LIN {X 0,Y 466.836,Z 671.645,A -85,B 0,C 180,E1 -7453.379,E2 -7453.379} C_VEL
LIN {X 0,Y 466.685,Z 675.645,A -85,B 0,C 180,E1 -7455.167,E2 -7455.167} C_VEL
LIN {X 0,Y 466.581,Z 678.329,A -85,B 0,C 180,E1 -7456.942,E2 -7456.942} C_VEL
LIN {X 0,Y 466.634,Z 679.796,A -85,B 0,C 180,E1 -7458.709,E2 -7458.709} C_VEL
LIN {X 0,Y 466.526,Z 680.097,A -85,B 0,C 180,E1 -7460.462,E2 -7460.462} C_VEL
LIN {X 0,Y 466.617,Z 679.249,A -85,B 0,C 180,E1 -7462.209,E2 -7462.209} C_VEL
LIN {X 0,Y 466.715,Z 677.258,A -85,B 0,C 180,E1 -7463.949,E2 -7463.949} C_VEL
LIN {X 0,Y 466.749,Z 674.056,A -85,B 0,C 180,E1 -7465.682,E2 -7465.682} C_VEL
LIN {X 0,Y 466.9,Z 669.606,A -85,B 0,C 180,E1 -7467.412,E2 -7467.412} C_VEL
LIN {X 0,Y 467.072,Z 663.846,A -85,B 0,C 180,E1 -7469.138,E2 -7469.138} C_VEL
LIN {X 0,Y 467.548,Z 656.595,A -85,B 0,C 180,E1 -7470.861,E2 -7470.861} C_VEL
LIN {X 0,Y 468.02,Z 648.866,A -85,B 0,C 180,E1 -7472.367,E2 -7472.367} C_VEL
LIN {X 0,Y 468.636,Z 639.619,A -85,B 0,C 180,E1 -7473.87,E2 -7473.87} C_VEL
LIN {X 0,Y 469.386,Z 628.509,A -85,B 0,C 180,E1 -7475.37,E2 -7475.37} C_VEL
LIN {X 0,Y 470.228,Z 617.061,A -85,B 0,C 180,E1 -7476.652,E2 -7476.652} C_VEL
LIN {X 0,Y 471.05,Z 604.485,A -85,B 0,C 180,E1 -7477.825,E2 -7477.825} C_VEL
LIN {X 0,Y 471.8,Z 592.099,A -85,B 0,C 180,E1 -7478.783,E2 -7478.783} C_VEL
LIN {X 0,Y 472.61,Z 578.629,A -85,B 0,C 180,E1 -7479.631,E2 -7479.631} C_VEL
LIN {X 0,Y 473.245,Z 564.922,A -85,B 0,C 180,E1 -7480.32,E2 -7480.32} C_VEL
LIN {X 0,Y 473.842,Z 550.313,A -85,B 0,C 180,E1 -7480.874,E2 -7480.874} C_VEL
LIN {X 0,Y 474.193,Z 534.838,A -85,B 0,C 180,E1 -7481.283,E2 -7481.283} C_VEL
LIN {X 0,Y 475.918,Z 391.809,A -85,B 0,C 180,E1 -7483.504,E2 -7483.504} C_VEL
LIN {X 0,Y 474.348,Z 384.081,A -85,B 0,C 180,E1 -7483.706,E2 -7483.706} C_VEL
LIN {X 0,Y 470.987,Z 371.045,A -85,B 0,C 180,E1 -7484.086,E2 -7484.086} C_VEL
LIN {X 0,Y 470.786,Z 370.175,A -85,B 0,C 180,E1 -7484.17,E2 -7484.17} C_VEL
LIN {X 0,Y 467.598,Z 355.867,A -85,B 0,C 180,E1 -7486.874,E2 -7486.874} C_VEL
LIN {X 0,Y 467.625,Z 355.863,A -85,B 0,C 180,E1 -7489.308,E2 -7489.308} C_VEL
LIN {X 0,Y 467.539,Z 355.872,A -85,B 0,C 180,E1 -7492.074,E2 -7492.074} C_VEL
LIN {X 0,Y 467.565,Z 355.866,A -85,B 0,C 180,E1 -7494.89,E2 -7494.89} C_VEL
LIN {X 0,Y 467.551,Z 355.872,A -85,B 0,C 180,E1 -7497.774,E2 -7497.774} C_VEL
LIN {X 0,Y 467.57,Z 355.865,A -85,B 0,C 180,E1 -7501.044,E2 -7501.044} C_VEL
LIN {X 0,Y 467.59,Z 355.862,A -85,B 0,C 180,E1 -7504.241,E2 -7504.241} C_VEL
LIN {X 0,Y 467.522,Z 355.869,A -85,B 0,C 180,E1 -7507.181,E2 -7507.181} C_VEL
LIN {X 0,Y 467.56,Z 355.859,A -85,B 0,C 180,E1 -7510.267,E2 -7510.267} C_VEL
LIN {X 0,Y 467.548,Z 355.87,A -85,B 0,C 180,E1 -7513.746,E2 -7513.746} C_VEL
LIN {X 0,Y 467.55,Z 355.86,A -85,B 0,C 180,E1 -7516.254,E2 -7516.254} C_VEL
LIN {X 0,Y 467.569,Z 355.864,A -85,B 0,C 180,E1 -7518.725,E2 -7518.725} C_VEL
LIN {X 0,Y 467.547,Z 355.869,A -85,B 0,C 180,E1 -7521.953,E2 -7521.953} C_VEL
LIN {X 0,Y 467.559,Z 355.868,A -85,B 0,C 180,E1 -7525.166,E2 -7525.166} C_VEL
LIN {X 0,Y 467.582,Z 355.864,A -85,B 0,C 180,E1 -7528.259,E2 -7528.259} C_VEL
LIN {X 0,Y 467.552,Z 355.866,A -85,B 0,C 180,E1 -7531.248,E2 -7531.248} C_VEL
LIN {X 0,Y 467.579,Z 355.843,A -85,B 0,C 180,E1 -7534.401,E2 -7534.401} C_VEL
LIN {X 0,Y 467.579,Z 355.857,A -85,B 0,C 180,E1 -7536.995,E2 -7536.995} C_VEL
LIN {X 0,Y 467.625,Z 355.861,A -85,B 0,C 180,E1 -7539.777,E2 -7539.777} C_VEL
LIN {X 0,Y 467.598,Z 355.852,A -85,B 0,C 180,E1 -7542.506,E2 -7542.506} C_VEL
LIN {X 0,Y 467.604,Z 355.861,A -85,B 0,C 180,E1 -7545.196,E2 -7545.196} C_VEL
LIN {X 0,Y 467.659,Z 355.848,A -85,B 0,C 180,E1 -7547.854,E2 -7547.854} C_VEL
LIN {X 0,Y 467.66,Z 355.855,A -85,B 0,C 180,E1 -7551.356,E2 -7551.356} C_VEL
LIN {X 0,Y 467.706,Z 355.842,A -85,B 0,C 180,E1 -7553.962,E2 -7553.962} C_VEL
LIN {X 0,Y 467.817,Z 355.835,A -85,B 0,C 180,E1 -7557.416,E2 -7557.416} C_VEL
LIN {X 0,Y 467.855,Z 355.826,A -85,B 0,C 180,E1 -7560,E2 -7560} C_VEL
LIN {X 0,Y 467.851,Z 355.824,A -85,B 0,C 180,E1 -7562.583,E2 -7562.583} C_VEL
LIN {X 0,Y 467.707,Z 355.847,A -85,B 0,C 180,E1 -7566.037,E2 -7566.037} C_VEL
LIN {X 0,Y 467.669,Z 355.847,A -85,B 0,C 180,E1 -7568.643,E2 -7568.643} C_VEL
LIN {X 0,Y 467.658,Z 355.849,A -85,B 0,C 180,E1 -7572.145,E2 -7572.145} C_VEL
LIN {X 0,Y 467.614,Z 355.863,A -85,B 0,C 180,E1 -7575.696,E2 -7575.696} C_VEL
LIN {X 0,Y 467.621,Z 355.857,A -85,B 0,C 180,E1 -7579.308,E2 -7579.308} C_VEL
LIN {X 0,Y 467.535,Z 355.866,A -85,B 0,C 180,E1 -7582.073,E2 -7582.073} C_VEL
LIN {X 0,Y 467.568,Z 355.863,A -85,B 0,C 180,E1 -7584.889,E2 -7584.889} C_VEL
LIN {X 0,Y 467.576,Z 355.869,A -85,B 0,C 180,E1 -7587.772,E2 -7587.772} C_VEL
LIN {X 0,Y 467.566,Z 355.865,A -85,B 0,C 180,E1 -7591.044,E2 -7591.044} C_VEL
LIN {X 0,Y 467.587,Z 355.863,A -85,B 0,C 180,E1 -7594.241,E2 -7594.241} C_VEL
LIN {X 0,Y 467.518,Z 355.872,A -85,B 0,C 180,E1 -7597.181,E2 -7597.181} C_VEL
LIN {X 0,Y 467.556,Z 355.865,A -85,B 0,C 180,E1 -7600.266,E2 -7600.266} C_VEL
LIN {X 0,Y 467.544,Z 355.873,A -85,B 0,C 180,E1 -7603.745,E2 -7603.745} C_VEL
LIN {X 0,Y 467.546,Z 355.869,A -85,B 0,C 180,E1 -7606.254,E2 -7606.254} C_VEL
LIN {X 0,Y 467.565,Z 355.866,A -85,B 0,C 180,E1 -7608.725,E2 -7608.725} C_VEL
LIN {X 0,Y 467.546,Z 355.871,A -85,B 0,C 180,E1 -7611.953,E2 -7611.953} C_VEL
LIN {X 0,Y 467.555,Z 355.87,A -85,B 0,C 180,E1 -7615.166,E2 -7615.166} C_VEL
LIN {X 0,Y 467.582,Z 355.866,A -85,B 0,C 180,E1 -7618.26,E2 -7618.26} C_VEL
LIN {X 0,Y 467.625,Z 356.033,A -85,B 0,C 180,E1 -7619.676,E2 -7619.676} C_VEL
LIN {X 0,Y 471.614,Z 372.945,A -85,B 0,C 180,E1 -7622.486,E2 -7622.486} C_VEL
LIN {X 0,Y 472.119,Z 377.049,A -85,B 0,C 180,E1 -7623.129,E2 -7623.129} C_VEL
LIN {X 0,Y 471.109,Z 396.315,A -85,B 0,C 180,E1 -7625.931,E2 -7625.931} C_VEL
LIN {X 0,Y 475.766,Z 421.055,A -85,B 0,C 180,E1 -7626.562,E2 -7626.562} C_VEL
LIN {X 0,Y 474.108,Z 562.68,A -85,B 0,C 180,E1 -7628.761,E2 -7628.761} C_VEL
LIN {X 0,Y 473.524,Z 578.617,A -85,B 0,C 180,E1 -7629.18,E2 -7629.18} C_VEL
LIN {X 0,Y 472.879,Z 594.115,A -85,B 0,C 180,E1 -7629.783,E2 -7629.783} C_VEL
LIN {X 0,Y 472.107,Z 608.851,A -85,B 0,C 180,E1 -7630.544,E2 -7630.544} C_VEL
LIN {X 0,Y 471.355,Z 622.223,A -85,B 0,C 180,E1 -7631.415,E2 -7631.415} C_VEL
LIN {X 0,Y 470.411,Z 635.801,A -85,B 0,C 180,E1 -7632.502,E2 -7632.502} C_VEL
LIN {X 0,Y 469.599,Z 648.146,A -85,B 0,C 180,E1 -7633.703,E2 -7633.703} C_VEL
LIN {X 0,Y 468.814,Z 659.403,A -85,B 0,C 180,E1 -7635.013,E2 -7635.013} C_VEL
LIN {X 0,Y 468.143,Z 670.327,A -85,B 0,C 180,E1 -7636.544,E2 -7636.544} C_VEL
LIN {X 0,Y 467.603,Z 679.411,A -85,B 0,C 180,E1 -7638.073,E2 -7638.073} C_VEL
LIN {X 0,Y 467.234,Z 686.944,A -85,B 0,C 180,E1 -7639.601,E2 -7639.601} C_VEL
LIN {X 0,Y 466.935,Z 693.971,A -85,B 0,C 180,E1 -7641.343,E2 -7641.343} C_VEL
LIN {X 0,Y 466.818,Z 699.495,A -85,B 0,C 180,E1 -7643.082,E2 -7643.082} C_VEL
LIN {X 0,Y 466.686,Z 703.668,A -85,B 0,C 180,E1 -7644.816,E2 -7644.816} C_VEL
LIN {X 0,Y 466.671,Z 706.594,A -85,B 0,C 180,E1 -7646.546,E2 -7646.546} C_VEL
LIN {X 0,Y 466.628,Z 708.336,A -85,B 0,C 180,E1 -7648.274,E2 -7648.274} C_VEL
LIN {X 0,Y 466.595,Z 708.93,A -85,B 0,C 180,E1 -7650,E2 -7650} C_VEL
LIN {X 0,Y 466.628,Z 708.325,A -85,B 0,C 180,E1 -7651.726,E2 -7651.726} C_VEL
LIN {X 0,Y 466.671,Z 706.573,A -85,B 0,C 180,E1 -7653.454,E2 -7653.454} C_VEL
LIN {X 0,Y 466.684,Z 703.644,A -85,B 0,C 180,E1 -7655.184,E2 -7655.184} C_VEL
LIN {X 0,Y 466.74,Z 699.47,A -85,B 0,C 180,E1 -7656.919,E2 -7656.919} C_VEL
LIN {X 0,Y 466.934,Z 693.945,A -85,B 0,C 180,E1 -7658.657,E2 -7658.657} C_VEL
LIN {X 0,Y 467.234,Z 686.922,A -85,B 0,C 180,E1 -7660.399,E2 -7660.399} C_VEL
LIN {X 0,Y 467.633,Z 679.411,A -85,B 0,C 180,E1 -7661.926,E2 -7661.926} C_VEL
LIN {X 0,Y 468.135,Z 670.368,A -85,B 0,C 180,E1 -7663.456,E2 -7663.456} C_VEL
LIN {X 0,Y 468.843,Z 659.518,A -85,B 0,C 180,E1 -7664.986,E2 -7664.986} C_VEL
LIN {X 0,Y 469.735,Z 647.346,A -85,B 0,C 180,E1 -7666.404,E2 -7666.404} C_VEL
LIN {X 0,Y 470.532,Z 634.953,A -85,B 0,C 180,E1 -7667.605,E2 -7667.605} C_VEL
LIN {X 0,Y 471.468,Z 621.272,A -85,B 0,C 180,E1 -7668.693,E2 -7668.693} C_VEL
LIN {X 0,Y 472.291,Z 607.87,A -85,B 0,C 180,E1 -7669.561,E2 -7669.561} C_VEL
LIN {X 0,Y 473.095,Z 593.523,A -85,B 0,C 180,E1 -7670.298,E2 -7670.298} C_VEL
LIN {X 0,Y 473.713,Z 578.414,A -85,B 0,C 180,E1 -7670.887,E2 -7670.887} C_VEL
LIN {X 0,Y 474.286,Z 562.15,A -85,B 0,C 180,E1 -7671.316,E2 -7671.316} C_VEL
LIN {X 0,Y 476.029,Z 420.259,A -85,B 0,C 180,E1 -7673.546,E2 -7673.546} C_VEL
LIN {X 0,Y 471.305,Z 396.045,A -85,B 0,C 180,E1 -7674.228,E2 -7674.228} C_VEL
LIN {X 0,Y 472.463,Z 377.157,A -85,B 0,C 180,E1 -7677.034,E2 -7677.034} C_VEL
LIN {X 0,Y 471.018,Z 369.489,A -85,B 0,C 180,E1 -7678.318,E2 -7678.318} C_VEL
LIN {X 0,Y 467.576,Z 355.874,A -85,B 0,C 180,E1 -7680.733,E2 -7680.733} C_VEL
LIN {X 0,Y 467.568,Z 355.869,A -85,B 0,C 180,E1 -7683.79,E2 -7683.79} C_VEL
LIN {X 0,Y 467.517,Z 355.874,A -85,B 0,C 180,E1 -7686.963,E2 -7686.963} C_VEL
LIN {X 0,Y 467.557,Z 355.87,A -85,B 0,C 180,E1 -7690.267,E2 -7690.267} C_VEL
LIN {X 0,Y 467.542,Z 355.869,A -85,B 0,C 180,E1 -7692.566,E2 -7692.566} C_VEL
LIN {X 0,Y 467.564,Z 355.867,A -85,B 0,C 180,E1 -7695.053,E2 -7695.053} C_VEL
LIN {X 0,Y 467.56,Z 355.87,A -85,B 0,C 180,E1 -7698.726,E2 -7698.726} C_VEL
LIN {X 0,Y 467.543,Z 355.87,A -85,B 0,C 180,E1 -7701.954,E2 -7701.954} C_VEL
LIN {X 0,Y 467.561,Z 355.863,A -85,B 0,C 180,E1 -7705.167,E2 -7705.167} C_VEL
LIN {X 0,Y 467.582,Z 355.857,A -85,B 0,C 180,E1 -7708.26,E2 -7708.26} C_VEL
LIN {X 0,Y 467.555,Z 355.864,A -85,B 0,C 180,E1 -7711.249,E2 -7711.249} C_VEL
LIN {X 0,Y 467.582,Z 355.863,A -85,B 0,C 180,E1 -7714.159,E2 -7714.159} C_VEL
LIN {X 0,Y 467.576,Z 355.862,A -85,B 0,C 180,E1 -7716.996,E2 -7716.996} C_VEL
LIN {X 0,Y 467.621,Z 355.858,A -85,B 0,C 180,E1 -7719.777,E2 -7719.777} C_VEL
LIN {X 0,Y 467.589,Z 355.867,A -85,B 0,C 180,E1 -7722.506,E2 -7722.506} C_VEL
LIN {X 0,Y 467.6,Z 355.86,A -85,B 0,C 180,E1 -7725.197,E2 -7725.197} C_VEL
LIN {X 0,Y 467.658,Z 355.851,A -85,B 0,C 180,E1 -7727.855,E2 -7727.855} C_VEL
LIN {X 0,Y 467.668,Z 355.848,A -85,B 0,C 180,E1 -7731.357,E2 -7731.357} C_VEL
LIN {X 0,Y 467.714,Z 355.848,A -85,B 0,C 180,E1 -7733.963,E2 -7733.963} C_VEL
LIN {X 0,Y 467.852,Z 355.829,A -85,B 0,C 180,E1 -7737.417,E2 -7737.417} C_VEL
LIN {X 0,Y 467.854,Z 355.826,A -85,B 0,C 180,E1 -7740,E2 -7740} C_VEL
LIN {X 0,Y 467.848,Z 355.831,A -85,B 0,C 180,E1 -7742.583,E2 -7742.583} C_VEL
LIN {X 0,Y 467.714,Z 355.849,A -85,B 0,C 180,E1 -7746.038,E2 -7746.038} C_VEL
LIN {X 0,Y 467.666,Z 355.858,A -85,B 0,C 180,E1 -7748.643,E2 -7748.643} C_VEL
LIN {X 0,Y 467.659,Z 355.854,A -85,B 0,C 180,E1 -7752.146,E2 -7752.146} C_VEL
LIN {X 0,Y 467.642,Z 355.854,A -85,B 0,C 180,E1 -7755.695,E2 -7755.695} C_VEL
LIN {X 0,Y 467.624,Z 355.843,A -85,B 0,C 180,E1 -7759.308,E2 -7759.308} C_VEL
LIN {X 0,Y 467.538,Z 355.868,A -85,B 0,C 180,E1 -7762.074,E2 -7762.074} C_VEL
LIN {X 0,Y 467.563,Z 355.856,A -85,B 0,C 180,E1 -7764.89,E2 -7764.89} C_VEL
LIN {X 0,Y 467.582,Z 355.862,A -85,B 0,C 180,E1 -7767.772,E2 -7767.772} C_VEL
LIN {X 0,Y 467.571,Z 355.857,A -85,B 0,C 180,E1 -7771.045,E2 -7771.045} C_VEL
LIN {X 0,Y 467.58,Z 355.868,A -85,B 0,C 180,E1 -7774.24,E2 -7774.24} C_VEL
LIN {X 0,Y 467.526,Z 355.872,A -85,B 0,C 180,E1 -7777.182,E2 -7777.182} C_VEL
LIN {X 0,Y 467.561,Z 355.865,A -85,B 0,C 180,E1 -7780.267,E2 -7780.267} C_VEL
LIN {X 0,Y 467.55,Z 355.869,A -85,B 0,C 180,E1 -7783.746,E2 -7783.746} C_VEL
LIN {X 0,Y 467.552,Z 355.869,A -85,B 0,C 180,E1 -7786.255,E2 -7786.255} C_VEL
LIN {X 0,Y 467.574,Z 355.867,A -85,B 0,C 180,E1 -7789.735,E2 -7789.735} C_VEL
LIN {X 0,Y 467.565,Z 355.969,A -85,B 0,C 180,E1 -7792.929,E2 -7792.929} C_VEL
LIN {X 0,Y 470.544,Z 368.645,A -85,B 0,C 180,E1 -7795.419,E2 -7795.419} C_VEL
LIN {X 0,Y 470.999,Z 370.7,A -85,B 0,C 180,E1 -7795.813,E2 -7795.813} C_VEL
LIN {X 0,Y 473.185,Z 377.561,A -85,B 0,C 180,E1 -7796.064,E2 -7796.064} C_VEL
LIN {X 0,Y 476.317,Z 391.74,A -85,B 0,C 180,E1 -7796.479,E2 -7796.479} C_VEL
LIN {X 0,Y 474.65,Z 517.95,A -85,B 0,C 180,E1 -7798.444,E2 -7798.444} C_VEL
LIN {X 0,Y 473.931,Z 523.804,A -85,B 0,C 180,E1 -7798.5,E2 -7798.5} C_VEL
LIN {X 0,Y 468.73,Z 540.884,A -85,B 0,C 180,E1 -7798.579,E2 -7798.579} C_VEL
LIN {X 0,Y 467.607,Z 546.618,A -85,B 0,C 180,E1 -7798.686,E2 -7798.686} C_VEL
LIN {X 0,Y 467.497,Z 548.534,A -85,B 0,C 180,E1 -7798.742,E2 -7798.742} C_VEL
LIN {X 0,Y 466.936,Z 563.073,A -85,B 0,C 180,E1 -7799.283,E2 -7799.283} C_VEL
LIN {X 0,Y 466.171,Z 577.184,A -85,B 0,C 180,E1 -7799.978,E2 -7799.978} C_VEL
LIN {X 0,Y 465.384,Z 591.094,A -85,B 0,C 180,E1 -7800.855,E2 -7800.855} C_VEL
LIN {X 0,Y 464.463,Z 604.731,A -85,B 0,C 180,E1 -7801.919,E2 -7801.919} C_VEL
LIN {X 0,Y 463.464,Z 617.402,A -85,B 0,C 180,E1 -7803.124,E2 -7803.124} C_VEL
LIN {X 0,Y 462.676,Z 628.129,A -85,B 0,C 180,E1 -7804.347,E2 -7804.347} C_VEL
LIN {X 0,Y 461.84,Z 638.445,A -85,B 0,C 180,E1 -7805.741,E2 -7805.741} C_VEL
LIN {X 0,Y 461.203,Z 647.16,A -85,B 0,C 180,E1 -7807.134,E2 -7807.134} C_VEL
LIN {X 0,Y 460.644,Z 655.619,A -85,B 0,C 180,E1 -7808.755,E2 -7808.755} C_VEL
LIN {X 0,Y 460.167,Z 662.538,A -85,B 0,C 180,E1 -7810.367,E2 -7810.367} C_VEL
LIN {X 0,Y 459.897,Z 668.876,A -85,B 0,C 180,E1 -7812.204,E2 -7812.204} C_VEL
LIN {X 0,Y 459.73,Z 673.684,A -85,B 0,C 180,E1 -7814.028,E2 -7814.028} C_VEL
LIN {X 0,Y 459.526,Z 677.12,A -85,B 0,C 180,E1 -7815.836,E2 -7815.836} C_VEL
LIN {X 0,Y 459.522,Z 679.296,A -85,B 0,C 180,E1 -7817.636,E2 -7817.636} C_VEL
LIN {X 0,Y 459.492,Z 680.282,A -85,B 0,C 180,E1 -7819.424,E2 -7819.424} C_VEL
LIN {X 0,Y 459.457,Z 680.115,A -85,B 0,C 180,E1 -7821.201,E2 -7821.201} C_VEL
LIN {X 0,Y 459.573,Z 678.794,A -85,B 0,C 180,E1 -7822.973,E2 -7822.973} C_VEL
LIN {X 0,Y 459.642,Z 676.271,A -85,B 0,C 180,E1 -7824.736,E2 -7824.736} C_VEL
LIN {X 0,Y 459.799,Z 672.548,A -85,B 0,C 180,E1 -7826.495,E2 -7826.495} C_VEL
LIN {X 0,Y 459.844,Z 667.581,A -85,B 0,C 180,E1 -7828.248,E2 -7828.248} C_VEL
LIN {X 0,Y 460.263,Z 661.209,A -85,B 0,C 180,E1 -7830,E2 -7830} C_VEL
LIN {X 0,Y 460.738,Z 653.281,A -85,B 0,C 180,E1 -7831.748,E2 -7831.748} C_VEL
LIN {X 0,Y 461.37,Z 644.846,A -85,B 0,C 180,E1 -7833.275,E2 -7833.275} C_VEL
LIN {X 0,Y 462.046,Z 634.757,A -85,B 0,C 180,E1 -7834.799,E2 -7834.799} C_VEL
LIN {X 0,Y 462.806,Z 624.46,A -85,B 0,C 180,E1 -7836.102,E2 -7836.102} C_VEL
LIN {X 0,Y 463.689,Z 613.277,A -85,B 0,C 180,E1 -7837.293,E2 -7837.293} C_VEL
LIN {X 0,Y 464.494,Z 601.199,A -85,B 0,C 180,E1 -7838.374,E2 -7838.374} C_VEL
LIN {X 0,Y 465.4,Z 588.004,A -85,B 0,C 180,E1 -7839.343,E2 -7839.343} C_VEL
LIN {X 0,Y 466.146,Z 573.447,A -85,B 0,C 180,E1 -7840.204,E2 -7840.204} C_VEL
LIN {X 0,Y 466.792,Z 559.337,A -85,B 0,C 180,E1 -7840.848,E2 -7840.848} C_VEL
LIN {X 0,Y 467.353,Z 544.154,A -85,B 0,C 180,E1 -7841.356,E2 -7841.356} C_VEL
LIN {X 0,Y 467.695,Z 529.518,A -85,B 0,C 180,E1 -7841.677,E2 -7841.677} C_VEL
LIN {X 0,Y 469.285,Z 391.719,A -85,B 0,C 180,E1 -7843.836,E2 -7843.836} C_VEL
LIN {X 0,Y 464.953,Z 374.167,A -85,B 0,C 180,E1 -7844.345,E2 -7844.345} C_VEL
LIN {X 0,Y 463.682,Z 370.698,A -85,B 0,C 180,E1 -7844.481,E2 -7844.481} C_VEL
LIN {X 0,Y 460.55,Z 356.745,A -85,B 0,C 180,E1 -7847.14,E2 -7847.14} C_VEL
LIN {X 0,Y 460.572,Z 356.742,A -85,B 0,C 180,E1 -7849.615,E2 -7849.615} C_VEL
LIN {X 0,Y 460.515,Z 356.745,A -85,B 0,C 180,E1 -7852.429,E2 -7852.429} C_VEL
LIN {X 0,Y 460.539,Z 356.745,A -85,B 0,C 180,E1 -7855.793,E2 -7855.793} C_VEL
LIN {X 0,Y 460.525,Z 356.745,A -85,B 0,C 180,E1 -7859.232,E2 -7859.232} C_VEL
LIN {X 0,Y 460.535,Z 356.736,A -85,B 0,C 180,E1 -7862.284,E2 -7862.284} C_VEL
LIN {X 0,Y 460.508,Z 356.747,A -85,B 0,C 180,E1 -7865.446,E2 -7865.446} C_VEL
LIN {X 0,Y 460.497,Z 356.746,A -85,B 0,C 180,E1 -7868.889,E2 -7868.889} C_VEL
LIN {X 0,Y 460.506,Z 356.745,A -85,B 0,C 180,E1 -7871.598,E2 -7871.598} C_VEL
LIN {X 0,Y 460.515,Z 356.74,A -85,B 0,C 180,E1 -7874.589,E2 -7874.589} C_VEL
LIN {X 0,Y 460.495,Z 356.75,A -85,B 0,C 180,E1 -7877.815,E2 -7877.815} C_VEL
LIN {X 0,Y 460.514,Z 356.742,A -85,B 0,C 180,E1 -7880.135,E2 -7880.135} C_VEL
LIN {X 0,Y 460.469,Z 356.755,A -85,B 0,C 180,E1 -7883.469,E2 -7883.469} C_VEL
LIN {X 0,Y 460.52,Z 356.74,A -85,B 0,C 180,E1 -7886.674,E2 -7886.674} C_VEL
LIN {X 0,Y 460.51,Z 356.745,A -85,B 0,C 180,E1 -7889.759,E2 -7889.759} C_VEL
LIN {X 0,Y 460.494,Z 356.729,A -85,B 0,C 180,E1 -7892.751,E2 -7892.751} C_VEL
LIN {X 0,Y 460.52,Z 356.732,A -85,B 0,C 180,E1 -7895.666,E2 -7895.666} C_VEL
LIN {X 0,Y 460.525,Z 356.741,A -85,B 0,C 180,E1 -7898.578,E2 -7898.578} C_VEL
LIN {X 0,Y 460.588,Z 356.737,A -85,B 0,C 180,E1 -7901.31,E2 -7901.31} C_VEL
LIN {X 0,Y 460.608,Z 356.732,A -85,B 0,C 180,E1 -7904.059,E2 -7904.059} C_VEL
LIN {X 0,Y 460.613,Z 356.728,A -85,B 0,C 180,E1 -7907.665,E2 -7907.665} C_VEL
LIN {X 0,Y 460.612,Z 356.731,A -85,B 0,C 180,E1 -7911.223,E2 -7911.223} C_VEL
LIN {X 0,Y 460.672,Z 356.719,A -85,B 0,C 180,E1 -7913.869,E2 -7913.869} C_VEL
LIN {X 0,Y 460.761,Z 356.714,A -85,B 0,C 180,E1 -7917.377,E2 -7917.377} C_VEL
LIN {X 0,Y 460.824,Z 356.702,A -85,B 0,C 180,E1 -7920,E2 -7920} C_VEL
LIN {X 0,Y 460.791,Z 356.703,A -85,B 0,C 180,E1 -7922.622,E2 -7922.622} C_VEL
LIN {X 0,Y 460.673,Z 356.722,A -85,B 0,C 180,E1 -7926.13,E2 -7926.13} C_VEL
LIN {X 0,Y 460.619,Z 356.726,A -85,B 0,C 180,E1 -7928.776,E2 -7928.776} C_VEL
LIN {X 0,Y 460.599,Z 356.727,A -85,B 0,C 180,E1 -7932.435,E2 -7932.435} C_VEL
LIN {X 0,Y 460.558,Z 356.738,A -85,B 0,C 180,E1 -7935.978,E2 -7935.978} C_VEL
LIN {X 0,Y 460.568,Z 356.74,A -85,B 0,C 180,E1 -7939.615,E2 -7939.615} C_VEL
LIN {X 0,Y 460.511,Z 356.738,A -85,B 0,C 180,E1 -7942.428,E2 -7942.428} C_VEL
LIN {X 0,Y 460.536,Z 356.742,A -85,B 0,C 180,E1 -7945.793,E2 -7945.793} C_VEL
LIN {X 0,Y 460.521,Z 356.743,A -85,B 0,C 180,E1 -7948.235,E2 -7948.235} C_VEL
LIN {X 0,Y 460.52,Z 356.745,A -85,B 0,C 180,E1 -7951.282,E2 -7951.282} C_VEL
LIN {X 0,Y 460.529,Z 356.741,A -85,B 0,C 180,E1 -7954.504,E2 -7954.504} C_VEL
LIN {X 0,Y 460.483,Z 356.752,A -85,B 0,C 180,E1 -7957.625,E2 -7957.625} C_VEL
LIN {X 0,Y 460.515,Z 356.742,A -85,B 0,C 180,E1 -7961.013,E2 -7961.013} C_VEL
LIN {X 0,Y 460.51,Z 356.743,A -85,B 0,C 180,E1 -7964.589,E2 -7964.589} C_VEL
LIN {X 0,Y 460.49,Z 356.753,A -85,B 0,C 180,E1 -7967.815,E2 -7967.815} C_VEL
LIN {X 0,Y 460.51,Z 356.749,A -85,B 0,C 180,E1 -7970.135,E2 -7970.135} C_VEL
LIN {X 0,Y 460.465,Z 356.757,A -85,B 0,C 180,E1 -7973.469,E2 -7973.469} C_VEL
LIN {X 0,Y 460.519,Z 356.745,A -85,B 0,C 180,E1 -7976.674,E2 -7976.674} C_VEL
LIN {X 0,Y 460.556,Z 356.767,A -85,B 0,C 180,E1 -7979.351,E2 -7979.351} C_VEL
LIN {X 0,Y 464.667,Z 374.114,A -85,B 0,C 180,E1 -7982.284,E2 -7982.284} C_VEL
LIN {X 0,Y 465.272,Z 377.365,A -85,B 0,C 180,E1 -7982.811,E2 -7982.811} C_VEL
LIN {X 0,Y 464.289,Z 396.076,A -85,B 0,C 180,E1 -7985.579,E2 -7985.579} C_VEL
LIN {X 0,Y 469.164,Z 422.584,A -85,B 0,C 180,E1 -7986.263,E2 -7986.263} C_VEL
LIN {X 0,Y 467.421,Z 562.843,A -85,B 0,C 180,E1 -7988.471,E2 -7988.471} C_VEL
LIN {X 0,Y 466.819,Z 578.838,A -85,B 0,C 180,E1 -7988.904,E2 -7988.904} C_VEL
LIN {X 0,Y 466.169,Z 593.903,A -85,B 0,C 180,E1 -7989.498,E2 -7989.498} C_VEL
LIN {X 0,Y 465.368,Z 608.345,A -85,B 0,C 180,E1 -7990.25,E2 -7990.25} C_VEL
LIN {X 0,Y 464.533,Z 621.77,A -85,B 0,C 180,E1 -7991.132,E2 -7991.132} C_VEL
LIN {X 0,Y 463.564,Z 635.41,A -85,B 0,C 180,E1 -7992.235,E2 -7992.235} C_VEL
LIN {X 0,Y 462.727,Z 647.794,A -85,B 0,C 180,E1 -7993.454,E2 -7993.454} C_VEL
LIN {X 0,Y 461.881,Z 659.078,A -85,B 0,C 180,E1 -7994.783,E2 -7994.783} C_VEL
LIN {X 0,Y 461.167,Z 670.036,A -85,B 0,C 180,E1 -7996.337,E2 -7996.337} C_VEL
LIN {X 0,Y 460.58,Z 679.136,A -85,B 0,C 180,E1 -7997.889,E2 -7997.889} C_VEL
LIN {X 0,Y 460.213,Z 686.683,A -85,B 0,C 180,E1 -7999.441,E2 -7999.441} C_VEL
LIN {X 0,Y 459.873,Z 693.725,A -85,B 0,C 180,E1 -8001.209,E2 -8001.209} C_VEL
LIN {X 0,Y 459.727,Z 699.259,A -85,B 0,C 180,E1 -8002.975,E2 -8002.975} C_VEL
LIN {X 0,Y 459.597,Z 703.44,A -85,B 0,C 180,E1 -8004.736,E2 -8004.736} C_VEL
LIN {X 0,Y 459.565,Z 706.37,A -85,B 0,C 180,E1 -8006.493,E2 -8006.493} C_VEL
LIN {X 0,Y 459.539,Z 708.116,A -85,B 0,C 180,E1 -8008.247,E2 -8008.247} C_VEL
LIN {X 0,Y 459.527,Z 708.712,A -85,B 0,C 180,E1 -8010,E2 -8010} C_VEL
LIN {X 0,Y 459.539,Z 708.108,A -85,B 0,C 180,E1 -8011.753,E2 -8011.753} C_VEL
LIN {X 0,Y 459.565,Z 706.358,A -85,B 0,C 180,E1 -8013.507,E2 -8013.507} C_VEL
LIN {X 0,Y 459.594,Z 703.433,A -85,B 0,C 180,E1 -8015.264,E2 -8015.264} C_VEL
LIN {X 0,Y 459.662,Z 699.265,A -85,B 0,C 180,E1 -8017.026,E2 -8017.026} C_VEL
LIN {X 0,Y 459.872,Z 693.751,A -85,B 0,C 180,E1 -8018.791,E2 -8018.791} C_VEL
LIN {X 0,Y 460.212,Z 686.741,A -85,B 0,C 180,E1 -8020.559,E2 -8020.559} C_VEL
LIN {X 0,Y 460.604,Z 679.242,A -85,B 0,C 180,E1 -8022.111,E2 -8022.111} C_VEL
LIN {X 0,Y 461.155,Z 670.22,A -85,B 0,C 180,E1 -8023.664,E2 -8023.664} C_VEL
LIN {X 0,Y 461.903,Z 659.397,A -85,B 0,C 180,E1 -8025.216,E2 -8025.216} C_VEL
LIN {X 0,Y 462.873,Z 647.272,A -85,B 0,C 180,E1 -8026.654,E2 -8026.654} C_VEL
LIN {X 0,Y 463.721,Z 634.921,A -85,B 0,C 180,E1 -8027.873,E2 -8027.873} C_VEL
LIN {X 0,Y 464.729,Z 621.305,A -85,B 0,C 180,E1 -8028.974,E2 -8028.974} C_VEL
LIN {X 0,Y 465.602,Z 607.964,A -85,B 0,C 180,E1 -8029.854,E2 -8029.854} C_VEL
LIN {X 0,Y 466.498,Z 592.589,A -85,B 0,C 180,E1 -8030.653,E2 -8030.653} C_VEL
LIN {X 0,Y 467.18,Z 577.109,A -85,B 0,C 180,E1 -8031.251,E2 -8031.251} C_VEL
LIN {X 0,Y 467.756,Z 561.566,A -85,B 0,C 180,E1 -8031.657,E2 -8031.657} C_VEL
LIN {X 0,Y 469.597,Z 421.323,A -85,B 0,C 180,E1 -8033.892,E2 -8033.892} C_VEL
LIN {X 0,Y 464.555,Z 395.836,A -85,B 0,C 180,E1 -8034.63,E2 -8034.63} C_VEL
LIN {X 0,Y 465.693,Z 379.057,A -85,B 0,C 180,E1 -8037.162,E2 -8037.162} C_VEL
LIN {X 0,Y 463.951,Z 370.166,A -85,B 0,C 180,E1 -8038.686,E2 -8038.686} C_VEL
LIN {X 0,Y 461.136,Z 359.008,A -85,B 0,C 180,E1 -8040.701,E2 -8040.701} C_VEL
LIN {X 0,Y 460.535,Z 356.745,A -85,B 0,C 180,E1 -8041.128,E2 -8041.128} C_VEL
LIN {X 0,Y 460.521,Z 356.748,A -85,B 0,C 180,E1 -8044.504,E2 -8044.504} C_VEL
LIN {X 0,Y 460.491,Z 356.748,A -85,B 0,C 180,E1 -8047.624,E2 -8047.624} C_VEL
LIN {X 0,Y 460.517,Z 356.742,A -85,B 0,C 180,E1 -8051.013,E2 -8051.013} C_VEL
LIN {X 0,Y 460.51,Z 356.749,A -85,B 0,C 180,E1 -8054.589,E2 -8054.589} C_VEL
LIN {X 0,Y 460.478,Z 356.75,A -85,B 0,C 180,E1 -8057.814,E2 -8057.814} C_VEL
LIN {X 0,Y 460.509,Z 356.748,A -85,B 0,C 180,E1 -8060.136,E2 -8060.136} C_VEL
LIN {X 0,Y 460.465,Z 356.74,A -85,B 0,C 180,E1 -8063.47,E2 -8063.47} C_VEL
LIN {X 0,Y 460.529,Z 356.743,A -85,B 0,C 180,E1 -8066.675,E2 -8066.675} C_VEL
LIN {X 0,Y 460.506,Z 356.731,A -85,B 0,C 180,E1 -8069.76,E2 -8069.76} C_VEL
LIN {X 0,Y 460.533,Z 356.741,A -85,B 0,C 180,E1 -8072.754,E2 -8072.754} C_VEL
LIN {X 0,Y 460.521,Z 356.743,A -85,B 0,C 180,E1 -8075.667,E2 -8075.667} C_VEL
LIN {X 0,Y 460.522,Z 356.748,A -85,B 0,C 180,E1 -8078.579,E2 -8078.579} C_VEL
LIN {X 0,Y 460.584,Z 356.733,A -85,B 0,C 180,E1 -8081.311,E2 -8081.311} C_VEL
LIN {X 0,Y 460.586,Z 356.735,A -85,B 0,C 180,E1 -8084.059,E2 -8084.059} C_VEL
LIN {X 0,Y 460.611,Z 356.728,A -85,B 0,C 180,E1 -8087.666,E2 -8087.666} C_VEL
LIN {X 0,Y 460.619,Z 356.726,A -85,B 0,C 180,E1 -8091.224,E2 -8091.224} C_VEL
LIN {X 0,Y 460.679,Z 356.724,A -85,B 0,C 180,E1 -8093.87,E2 -8093.87} C_VEL
LIN {X 0,Y 460.792,Z 356.708,A -85,B 0,C 180,E1 -8097.378,E2 -8097.378} C_VEL
LIN {X 0,Y 460.824,Z 356.702,A -85,B 0,C 180,E1 -8100,E2 -8100} C_VEL
LIN {X 0,Y 460.788,Z 356.71,A -85,B 0,C 180,E1 -8102.623,E2 -8102.623} C_VEL
LIN {X 0,Y 460.678,Z 356.726,A -85,B 0,C 180,E1 -8106.131,E2 -8106.131} C_VEL
LIN {X 0,Y 460.617,Z 356.734,A -85,B 0,C 180,E1 -8108.777,E2 -8108.777} C_VEL
LIN {X 0,Y 460.616,Z 356.735,A -85,B 0,C 180,E1 -8112.445,E2 -8112.445} C_VEL
LIN {X 0,Y 460.603,Z 356.733,A -85,B 0,C 180,E1 -8115.998,E2 -8115.998} C_VEL
LIN {X 0,Y 460.57,Z 356.721,A -85,B 0,C 180,E1 -8119.616,E2 -8119.616} C_VEL
LIN {X 0,Y 460.514,Z 356.748,A -85,B 0,C 180,E1 -8122.429,E2 -8122.429} C_VEL
LIN {X 0,Y 460.537,Z 356.728,A -85,B 0,C 180,E1 -8125.794,E2 -8125.794} C_VEL
LIN {X 0,Y 460.528,Z 356.744,A -85,B 0,C 180,E1 -8128.235,E2 -8128.235} C_VEL
LIN {X 0,Y 460.524,Z 356.735,A -85,B 0,C 180,E1 -8131.283,E2 -8131.283} C_VEL
LIN {X 0,Y 460.525,Z 356.741,A -85,B 0,C 180,E1 -8134.504,E2 -8134.504} C_VEL
LIN {X 0,Y 460.489,Z 356.747,A -85,B 0,C 180,E1 -8137.625,E2 -8137.625} C_VEL
LIN {X 0,Y 460.521,Z 356.745,A -85,B 0,C 180,E1 -8141.013,E2 -8141.013} C_VEL
LIN {X 0,Y 460.515,Z 356.746,A -85,B 0,C 180,E1 -8144.59,E2 -8144.59} C_VEL
LIN {X 0,Y 460.508,Z 356.743,A -85,B 0,C 180,E1 -8147.817,E2 -8147.817} C_VEL
LIN {X 0,Y 460.523,Z 356.748,A -85,B 0,C 180,E1 -8150.137,E2 -8150.137} C_VEL
LIN {X 0,Y 460.508,Z 356.834,A -85,B 0,C 180,E1 -8152.557,E2 -8152.557} C_VEL
LIN {X 0,Y 463.625,Z 369.899,A -85,B 0,C 180,E1 -8155.177,E2 -8155.177} C_VEL
LIN {X 0,Y 463.923,Z 371.197,A -85,B 0,C 180,E1 -8155.397,E2 -8155.397} C_VEL
LIN {X 0,Y 466.741,Z 378.624,A -85,B 0,C 180,E1 -8155.697,E2 -8155.697} C_VEL
LIN {X 0,Y 469.834,Z 392.084,A -85,B 0,C 180,E1 -8156.108,E2 -8156.108} C_VEL
LIN {X 0,Y 468.092,Z 520.515,A -85,B 0,C 180,E1 -8158.14,E2 -8158.14} C_VEL
LIN {X 0,Y 467.825,Z 539.358,A -85,B 0,C 180,E1 -8158.492,E2 -8158.492} C_VEL
LIN {X 0,Y 467.497,Z 548.534,A -85,B 0,C 180,E1 -8158.742,E2 -8158.742} C_VEL
LIN {X 0,Y 466.667,Z 554.254,A -85,B 0,C 180,E1 -8158.898,E2 -8158.898} C_VEL
LIN {X 0,Y 463.605,Z 563.513,A -85,B 0,C 180,E1 -8159.126,E2 -8159.126} C_VEL
LIN {X 0,Y 460.477,Z 572.639,A -85,B 0,C 180,E1 -8159.422,E2 -8159.422} C_VEL
LIN {X 0,Y 459.538,Z 578.009,A -85,B 0,C 180,E1 -8159.686,E2 -8159.686} C_VEL
LIN {X 0,Y 458.76,Z 591.001,A -85,B 0,C 180,E1 -8160.519,E2 -8160.519} C_VEL
LIN {X 0,Y 457.777,Z 604.5,A -85,B 0,C 180,E1 -8161.58,E2 -8161.58} C_VEL
LIN {X 0,Y 456.781,Z 616.656,A -85,B 0,C 180,E1 -8162.74,E2 -8162.74} C_VEL
LIN {X 0,Y 455.936,Z 627.219,A -85,B 0,C 180,E1 -8163.94,E2 -8163.94} C_VEL
LIN {X 0,Y 455.051,Z 637.721,A -85,B 0,C 180,E1 -8165.355,E2 -8165.355} C_VEL
LIN {X 0,Y 454.35,Z 646.543,A -85,B 0,C 180,E1 -8166.769,E2 -8166.769} C_VEL
LIN {X 0,Y 453.764,Z 654.697,A -85,B 0,C 180,E1 -8168.327,E2 -8168.327} C_VEL
LIN {X 0,Y 453.192,Z 662.174,A -85,B 0,C 180,E1 -8170.052,E2 -8170.052} C_VEL
LIN {X 0,Y 452.869,Z 668.633,A -85,B 0,C 180,E1 -8171.918,E2 -8171.918} C_VEL
LIN {X 0,Y 452.649,Z 673.558,A -85,B 0,C 180,E1 -8173.771,E2 -8173.771} C_VEL
LIN {X 0,Y 452.474,Z 677.104,A -85,B 0,C 180,E1 -8175.61,E2 -8175.61} C_VEL
LIN {X 0,Y 452.432,Z 679.387,A -85,B 0,C 180,E1 -8177.439,E2 -8177.439} C_VEL
LIN {X 0,Y 452.47,Z 680.076,A -85,B 0,C 180,E1 -8178.351,E2 -8178.351} C_VEL
LIN {X 0,Y 452.351,Z 680.588,A -85,B 0,C 180,E1 -8180.16,E2 -8180.16} C_VEL
LIN {X 0,Y 452.427,Z 679.926,A -85,B 0,C 180,E1 -8181.963,E2 -8181.963} C_VEL
LIN {X 0,Y 452.567,Z 678.075,A -85,B 0,C 180,E1 -8183.759,E2 -8183.759} C_VEL
LIN {X 0,Y 452.559,Z 675.069,A -85,B 0,C 180,E1 -8185.547,E2 -8185.547} C_VEL
LIN {X 0,Y 452.768,Z 670.833,A -85,B 0,C 180,E1 -8187.331,E2 -8187.331} C_VEL
LIN {X 0,Y 452.916,Z 665.302,A -85,B 0,C 180,E1 -8189.111,E2 -8189.111} C_VEL
LIN {X 0,Y 453.451,Z 658.292,A -85,B 0,C 180,E1 -8190.888,E2 -8190.888} C_VEL
LIN {X 0,Y 453.927,Z 650.832,A -85,B 0,C 180,E1 -8192.44,E2 -8192.44} C_VEL
LIN {X 0,Y 454.64,Z 641.876,A -85,B 0,C 180,E1 -8193.989,E2 -8193.989} C_VEL
LIN {X 0,Y 455.431,Z 631.112,A -85,B 0,C 180,E1 -8195.535,E2 -8195.535} C_VEL
LIN {X 0,Y 456.343,Z 620.071,A -85,B 0,C 180,E1 -8196.855,E2 -8196.855} C_VEL
LIN {X 0,Y 457.229,Z 607.992,A -85,B 0,C 180,E1 -8198.063,E2 -8198.063} C_VEL
LIN {X 0,Y 458.144,Z 594.728,A -85,B 0,C 180,E1 -8199.158,E2 -8199.158} C_VEL
LIN {X 0,Y 459.035,Z 581.695,A -85,B 0,C 180,E1 -8200.03,E2 -8200.03} C_VEL
LIN {X 0,Y 459.72,Z 568.569,A -85,B 0,C 180,E1 -8200.738,E2 -8200.738} C_VEL
LIN {X 0,Y 460.366,Z 554.247,A -85,B 0,C 180,E1 -8201.335,E2 -8201.335} C_VEL
LIN {X 0,Y 460.763,Z 538.764,A -85,B 0,C 180,E1 -8201.799,E2 -8201.799} C_VEL
LIN {X 0,Y 461.198,Z 517.405,A -85,B 0,C 180,E1 -8202.179,E2 -8202.179} C_VEL
LIN {X 0,Y 462.684,Z 392.58,A -85,B 0,C 180,E1 -8204.159,E2 -8204.159} C_VEL
LIN {X 0,Y 458.612,Z 376.375,A -85,B 0,C 180,E1 -8204.641,E2 -8204.641} C_VEL
LIN {X 0,Y 456.508,Z 370.839,A -85,B 0,C 180,E1 -8204.869,E2 -8204.869} C_VEL
LIN {X 0,Y 453.515,Z 357.622,A -85,B 0,C 180,E1 -8207.444,E2 -8207.444} C_VEL
LIN {X 0,Y 453.508,Z 357.618,A -85,B 0,C 180,E1 -8209.934,E2 -8209.934} C_VEL
LIN {X 0,Y 453.483,Z 357.622,A -85,B 0,C 180,E1 -8212.796,E2 -8212.796} C_VEL
LIN {X 0,Y 453.487,Z 357.621,A -85,B 0,C 180,E1 -8215.989,E2 -8215.989} C_VEL
LIN {X 0,Y 453.468,Z 357.621,A -85,B 0,C 180,E1 -8218.715,E2 -8218.715} C_VEL
LIN {X 0,Y 453.468,Z 357.621,A -85,B 0,C 180,E1 -8221.799,E2 -8221.799} C_VEL
LIN {X 0,Y 453.481,Z 357.621,A -85,B 0,C 180,E1 -8224.989,E2 -8224.989} C_VEL
LIN {X 0,Y 453.45,Z 357.623,A -85,B 0,C 180,E1 -8228.313,E2 -8228.313} C_VEL
LIN {X 0,Y 453.474,Z 357.613,A -85,B 0,C 180,E1 -8230.611,E2 -8230.611} C_VEL
LIN {X 0,Y 453.485,Z 357.616,A -85,B 0,C 180,E1 -8234.528,E2 -8234.528} C_VEL
LIN {X 0,Y 453.452,Z 357.624,A -85,B 0,C 180,E1 -8238.069,E2 -8238.069} C_VEL
LIN {X 0,Y 453.443,Z 357.621,A -85,B 0,C 180,E1 -8240.802,E2 -8240.802} C_VEL
LIN {X 0,Y 453.451,Z 357.625,A -85,B 0,C 180,E1 -8243.916,E2 -8243.916} C_VEL
LIN {X 0,Y 453.478,Z 357.62,A -85,B 0,C 180,E1 -8247.15,E2 -8247.15} C_VEL
LIN {X 0,Y 453.468,Z 357.617,A -85,B 0,C 180,E1 -8250.267,E2 -8250.267} C_VEL
LIN {X 0,Y 453.443,Z 357.604,A -85,B 0,C 180,E1 -8253.289,E2 -8253.289} C_VEL
LIN {X 0,Y 453.496,Z 357.61,A -85,B 0,C 180,E1 -8256.238,E2 -8256.238} C_VEL
LIN {X 0,Y 453.486,Z 357.62,A -85,B 0,C 180,E1 -8259.117,E2 -8259.117} C_VEL
LIN {X 0,Y 453.504,Z 357.611,A -85,B 0,C 180,E1 -8261.944,E2 -8261.944} C_VEL
LIN {X 0,Y 453.541,Z 357.61,A -85,B 0,C 180,E1 -8264.726,E2 -8264.726} C_VEL
LIN {X 0,Y 453.561,Z 357.599,A -85,B 0,C 180,E1 -8268.379,E2 -8268.379} C_VEL
LIN {X 0,Y 453.58,Z 357.606,A -85,B 0,C 180,E1 -8271.086,E2 -8271.086} C_VEL
LIN {X 0,Y 453.64,Z 357.596,A -85,B 0,C 180,E1 -8273.774,E2 -8273.774} C_VEL
LIN {X 0,Y 453.708,Z 357.592,A -85,B 0,C 180,E1 -8277.336,E2 -8277.336} C_VEL
LIN {X 0,Y 453.794,Z 357.577,A -85,B 0,C 180,E1 -8280,E2 -8280} C_VEL
LIN {X 0,Y 453.735,Z 357.582,A -85,B 0,C 180,E1 -8282.663,E2 -8282.663} C_VEL
LIN {X 0,Y 453.641,Z 357.597,A -85,B 0,C 180,E1 -8286.225,E2 -8286.225} C_VEL
LIN {X 0,Y 453.585,Z 357.602,A -85,B 0,C 180,E1 -8288.913,E2 -8288.913} C_VEL
LIN {X 0,Y 453.566,Z 357.603,A -85,B 0,C 180,E1 -8292.528,E2 -8292.528} C_VEL
LIN {X 0,Y 453.504,Z 357.615,A -85,B 0,C 180,E1 -8296.091,E2 -8296.091} C_VEL
LIN {X 0,Y 453.518,Z 357.611,A -85,B 0,C 180,E1 -8299.039,E2 -8299.039} C_VEL
LIN {X 0,Y 453.478,Z 357.619,A -85,B 0,C 180,E1 -8301.836,E2 -8301.836} C_VEL
LIN {X 0,Y 453.491,Z 357.616,A -85,B 0,C 180,E1 -8304.735,E2 -8304.735} C_VEL
LIN {X 0,Y 453.481,Z 357.622,A -85,B 0,C 180,E1 -8307.947,E2 -8307.947} C_VEL
LIN {X 0,Y 453.474,Z 357.619,A -85,B 0,C 180,E1 -8310.759,E2 -8310.759} C_VEL
LIN {X 0,Y 453.475,Z 357.624,A -85,B 0,C 180,E1 -8313.913,E2 -8313.913} C_VEL
LIN {X 0,Y 453.436,Z 357.627,A -85,B 0,C 180,E1 -8317.191,E2 -8317.191} C_VEL
LIN {X 0,Y 453.469,Z 357.619,A -85,B 0,C 180,E1 -8320.611,E2 -8320.611} C_VEL
LIN {X 0,Y 453.481,Z 357.619,A -85,B 0,C 180,E1 -8324.528,E2 -8324.528} C_VEL
LIN {X 0,Y 453.448,Z 357.628,A -85,B 0,C 180,E1 -8328.069,E2 -8328.069} C_VEL
LIN {X 0,Y 453.442,Z 357.627,A -85,B 0,C 180,E1 -8330.801,E2 -8330.801} C_VEL
LIN {X 0,Y 453.447,Z 357.627,A -85,B 0,C 180,E1 -8333.916,E2 -8333.916} C_VEL
LIN {X 0,Y 453.478,Z 357.624,A -85,B 0,C 180,E1 -8337.151,E2 -8337.151} C_VEL
LIN {X 0,Y 453.537,Z 357.742,A -85,B 0,C 180,E1 -8339.061,E2 -8339.061} C_VEL
LIN {X 0,Y 457.675,Z 375.263,A -85,B 0,C 180,E1 -8342.072,E2 -8342.072} C_VEL
LIN {X 0,Y 458.431,Z 379.494,A -85,B 0,C 180,E1 -8342.769,E2 -8342.769} C_VEL
LIN {X 0,Y 457.466,Z 395.864,A -85,B 0,C 180,E1 -8345.221,E2 -8345.221} C_VEL
LIN {X 0,Y 462.554,Z 422.526,A -85,B 0,C 180,E1 -8345.932,E2 -8345.932} C_VEL
LIN {X 0,Y 460.806,Z 559.95,A -85,B 0,C 180,E1 -8348.117,E2 -8348.117} C_VEL
LIN {X 0,Y 460.289,Z 575.317,A -85,B 0,C 180,E1 -8348.503,E2 -8348.503} C_VEL
LIN {X 0,Y 459.64,Z 590.167,A -85,B 0,C 180,E1 -8349.055,E2 -8349.055} C_VEL
LIN {X 0,Y 458.806,Z 604.801,A -85,B 0,C 180,E1 -8349.781,E2 -8349.781} C_VEL
LIN {X 0,Y 457.974,Z 618.074,A -85,B 0,C 180,E1 -8350.619,E2 -8350.619} C_VEL
LIN {X 0,Y 457.021,Z 631.08,A -85,B 0,C 180,E1 -8351.624,E2 -8351.624} C_VEL
LIN {X 0,Y 456.046,Z 643.957,A -85,B 0,C 180,E1 -8352.836,E2 -8352.836} C_VEL
LIN {X 0,Y 455.232,Z 655.121,A -85,B 0,C 180,E1 -8354.096,E2 -8354.096} C_VEL
LIN {X 0,Y 454.479,Z 665.234,A -85,B 0,C 180,E1 -8355.446,E2 -8355.446} C_VEL
LIN {X 0,Y 453.821,Z 673.953,A -85,B 0,C 180,E1 -8356.818,E2 -8356.818} C_VEL
LIN {X 0,Y 453.352,Z 683.344,A -85,B 0,C 180,E1 -8358.6,E2 -8358.6} C_VEL
LIN {X 0,Y 452.897,Z 690.129,A -85,B 0,C 180,E1 -8360.172,E2 -8360.172} C_VEL
LIN {X 0,Y 452.696,Z 696.412,A -85,B 0,C 180,E1 -8361.968,E2 -8361.968} C_VEL
LIN {X 0,Y 452.561,Z 701.266,A -85,B 0,C 180,E1 -8363.759,E2 -8363.759} C_VEL
LIN {X 0,Y 452.45,Z 704.821,A -85,B 0,C 180,E1 -8365.546,E2 -8365.546} C_VEL
LIN {X 0,Y 452.501,Z 707.162,A -85,B 0,C 180,E1 -8367.329,E2 -8367.329} C_VEL
LIN {X 0,Y 452.426,Z 708.339,A -85,B 0,C 180,E1 -8369.11,E2 -8369.11} C_VEL
LIN {X 0,Y 452.426,Z 708.337,A -85,B 0,C 180,E1 -8370.89,E2 -8370.89} C_VEL
LIN {X 0,Y 452.501,Z 707.167,A -85,B 0,C 180,E1 -8372.671,E2 -8372.671} C_VEL
LIN {X 0,Y 452.449,Z 704.84,A -85,B 0,C 180,E1 -8374.454,E2 -8374.454} C_VEL
LIN {X 0,Y 452.551,Z 701.097,A -85,B 0,C 180,E1 -8376.331,E2 -8376.331} C_VEL
LIN {X 0,Y 452.696,Z 696.503,A -85,B 0,C 180,E1 -8378.032,E2 -8378.032} C_VEL
LIN {X 0,Y 452.894,Z 690.274,A -85,B 0,C 180,E1 -8379.828,E2 -8379.828} C_VEL
LIN {X 0,Y 453.37,Z 683.538,A -85,B 0,C 180,E1 -8381.399,E2 -8381.399} C_VEL
LIN {X 0,Y 453.808,Z 675.666,A -85,B 0,C 180,E1 -8382.931,E2 -8382.931} C_VEL
LIN {X 0,Y 454.505,Z 665.698,A -85,B 0,C 180,E1 -8384.553,E2 -8384.553} C_VEL
LIN {X 0,Y 455.283,Z 655.783,A -85,B 0,C 180,E1 -8385.902,E2 -8385.902} C_VEL
LIN {X 0,Y 456.25,Z 644.049,A -85,B 0,C 180,E1 -8387.247,E2 -8387.247} C_VEL
LIN {X 0,Y 457.228,Z 631.075,A -85,B 0,C 180,E1 -8388.483,E2 -8388.483} C_VEL
LIN {X 0,Y 458.207,Z 618.237,A -85,B 0,C 180,E1 -8389.488,E2 -8389.488} C_VEL
LIN {X 0,Y 459.185,Z 604.232,A -85,B 0,C 180,E1 -8390.377,E2 -8390.377} C_VEL
LIN {X 0,Y 460.012,Z 590.164,A -85,B 0,C 180,E1 -8391.082,E2 -8391.082} C_VEL
LIN {X 0,Y 460.718,Z 574.944,A -85,B 0,C 180,E1 -8391.652,E2 -8391.652} C_VEL
LIN {X 0,Y 461.283,Z 559.673,A -85,B 0,C 180,E1 -8392.036,E2 -8392.036} C_VEL
LIN {X 0,Y 463.182,Z 422.438,A -85,B 0,C 180,E1 -8394.251,E2 -8394.251} C_VEL
LIN {X 0,Y 458.229,Z 397.446,A -85,B 0,C 180,E1 -8394.983,E2 -8394.983} C_VEL
LIN {X 0,Y 457.883,Z 395.611,A -85,B 0,C 180,E1 -8395.046,E2 -8395.046} C_VEL
LIN {X 0,Y 458.922,Z 380.632,A -85,B 0,C 180,E1 -8397.35,E2 -8397.35} C_VEL
LIN {X 0,Y 456.621,Z 369.584,A -85,B 0,C 180,E1 -8399.294,E2 -8399.294} C_VEL
LIN {X 0,Y 453.463,Z 357.627,A -85,B 0,C 180,E1 -8401.551,E2 -8401.551} C_VEL
LIN {X 0,Y 453.48,Z 357.624,A -85,B 0,C 180,E1 -8404.776,E2 -8404.776} C_VEL
LIN {X 0,Y 453.447,Z 357.624,A -85,B 0,C 180,E1 -8408.313,E2 -8408.313} C_VEL
LIN {X 0,Y 453.469,Z 357.623,A -85,B 0,C 180,E1 -8410.612,E2 -8410.612} C_VEL
LIN {X 0,Y 453.458,Z 357.627,A -85,B 0,C 180,E1 -8414.222,E2 -8414.222} C_VEL
LIN {X 0,Y 453.425,Z 357.628,A -85,B 0,C 180,E1 -8417.001,E2 -8417.001} C_VEL
LIN {X 0,Y 453.469,Z 357.621,A -85,B 0,C 180,E1 -8419.413,E2 -8419.413} C_VEL
LIN {X 0,Y 453.438,Z 357.618,A -85,B 0,C 180,E1 -8422.809,E2 -8422.809} C_VEL
LIN {X 0,Y 453.476,Z 357.621,A -85,B 0,C 180,E1 -8426.088,E2 -8426.088} C_VEL
LIN {X 0,Y 453.475,Z 357.605,A -85,B 0,C 180,E1 -8429.241,E2 -8429.241} C_VEL
LIN {X 0,Y 453.507,Z 357.621,A -85,B 0,C 180,E1 -8432.296,E2 -8432.296} C_VEL
LIN {X 0,Y 453.494,Z 357.618,A -85,B 0,C 180,E1 -8435.265,E2 -8435.265} C_VEL
LIN {X 0,Y 453.481,Z 357.625,A -85,B 0,C 180,E1 -8438.415,E2 -8438.415} C_VEL
LIN {X 0,Y 453.523,Z 357.614,A -85,B 0,C 180,E1 -8441.009,E2 -8441.009} C_VEL
LIN {X 0,Y 453.538,Z 357.612,A -85,B 0,C 180,E1 -8443.894,E2 -8443.894} C_VEL
LIN {X 0,Y 453.565,Z 357.605,A -85,B 0,C 180,E1 -8447.472,E2 -8447.472} C_VEL
LIN {X 0,Y 453.585,Z 357.603,A -85,B 0,C 180,E1 -8451.087,E2 -8451.087} C_VEL
LIN {X 0,Y 453.645,Z 357.6,A -85,B 0,C 180,E1 -8453.775,E2 -8453.775} C_VEL
LIN {X 0,Y 453.736,Z 357.587,A -85,B 0,C 180,E1 -8457.337,E2 -8457.337} C_VEL
LIN {X 0,Y 453.793,Z 357.577,A -85,B 0,C 180,E1 -8460,E2 -8460} C_VEL
LIN {X 0,Y 453.732,Z 357.588,A -85,B 0,C 180,E1 -8462.664,E2 -8462.664} C_VEL
LIN {X 0,Y 453.645,Z 357.604,A -85,B 0,C 180,E1 -8466.226,E2 -8466.226} C_VEL
LIN {X 0,Y 453.584,Z 357.609,A -85,B 0,C 180,E1 -8468.914,E2 -8468.914} C_VEL
LIN {X 0,Y 453.566,Z 357.615,A -85,B 0,C 180,E1 -8472.529,E2 -8472.529} C_VEL
LIN {X 0,Y 453.547,Z 357.614,A -85,B 0,C 180,E1 -8476.196,E2 -8476.196} C_VEL
LIN {X 0,Y 453.519,Z 357.6,A -85,B 0,C 180,E1 -8479.039,E2 -8479.039} C_VEL
LIN {X 0,Y 453.48,Z 357.617,A -85,B 0,C 180,E1 -8481.836,E2 -8481.836} C_VEL
LIN {X 0,Y 453.472,Z 357.612,A -85,B 0,C 180,E1 -8484.737,E2 -8484.737} C_VEL
LIN {X 0,Y 453.493,Z 357.618,A -85,B 0,C 180,E1 -8487.95,E2 -8487.95} C_VEL
LIN {X 0,Y 453.479,Z 357.612,A -85,B 0,C 180,E1 -8490.76,E2 -8490.76} C_VEL
LIN {X 0,Y 453.471,Z 357.623,A -85,B 0,C 180,E1 -8493.914,E2 -8493.914} C_VEL
LIN {X 0,Y 453.442,Z 357.626,A -85,B 0,C 180,E1 -8497.191,E2 -8497.191} C_VEL
LIN {X 0,Y 453.473,Z 357.625,A -85,B 0,C 180,E1 -8500.612,E2 -8500.612} C_VEL
LIN {X 0,Y 453.462,Z 357.627,A -85,B 0,C 180,E1 -8504.222,E2 -8504.222} C_VEL
LIN {X 0,Y 453.452,Z 357.625,A -85,B 0,C 180,E1 -8507.004,E2 -8507.004} C_VEL
LIN {X 0,Y 453.497,Z 357.621,A -85,B 0,C 180,E1 -8509.409,E2 -8509.409} C_VEL
LIN {X 0,Y 453.479,Z 357.783,A -85,B 0,C 180,E1 -8512.186,E2 -8512.186} C_VEL
LIN {X 0,Y 456.76,Z 371.28,A -85,B 0,C 180,E1 -8514.943,E2 -8514.943} C_VEL
LIN {X 0,Y 460.574,Z 380.684,A -85,B 0,C 180,E1 -8515.349,E2 -8515.349} C_VEL
LIN {X 0,Y 463.467,Z 393.384,A -85,B 0,C 180,E1 -8515.747,E2 -8515.747} C_VEL
LIN {X 0,Y 461.499,Z 525.089,A -85,B 0,C 180,E1 -8517.856,E2 -8517.856} C_VEL
LIN {X 0,Y 461.303,Z 540.868,A -85,B 0,C 180,E1 -8518.179,E2 -8518.179} C_VEL
LIN {X 0,Y 460.757,Z 555.289,A -85,B 0,C 180,E1 -8518.625,E2 -8518.625} C_VEL
LIN {X 0,Y 459.989,Z 570.38,A -85,B 0,C 180,E1 -8519.278,E2 -8519.278} C_VEL
LIN {X 0,Y 459.538,Z 578.009,A -85,B 0,C 180,E1 -8519.686,E2 -8519.686} C_VEL
LIN {X 0,Y 458.583,Z 583.4,A -85,B 0,C 180,E1 -8519.973,E2 -8519.973} C_VEL
LIN {X 0,Y 455.329,Z 592.054,A -85,B 0,C 180,E1 -8520.421,E2 -8520.421} C_VEL
LIN {X 0,Y 452.035,Z 600.491,A -85,B 0,C 180,E1 -8520.936,E2 -8520.936} C_VEL
LIN {X 0,Y 451.029,Z 605.377,A -85,B 0,C 180,E1 -8521.327,E2 -8521.327} C_VEL
LIN {X 0,Y 449.939,Z 617.964,A -85,B 0,C 180,E1 -8522.563,E2 -8522.563} C_VEL
LIN {X 0,Y 449.049,Z 628.19,A -85,B 0,C 180,E1 -8523.76,E2 -8523.76} C_VEL
LIN {X 0,Y 448.064,Z 639.199,A -85,B 0,C 180,E1 -8525.295,E2 -8525.295} C_VEL
LIN {X 0,Y 447.245,Z 648.588,A -85,B 0,C 180,E1 -8526.868,E2 -8526.868} C_VEL
LIN {X 0,Y 446.674,Z 656.518,A -85,B 0,C 180,E1 -8528.462,E2 -8528.462} C_VEL
LIN {X 0,Y 446.089,Z 663.661,A -85,B 0,C 180,E1 -8530.201,E2 -8530.201} C_VEL
LIN {X 0,Y 445.764,Z 669.836,A -85,B 0,C 180,E1 -8532.095,E2 -8532.095} C_VEL
LIN {X 0,Y 445.592,Z 673.442,A -85,B 0,C 180,E1 -8533.507,E2 -8533.507} C_VEL
LIN {X 0,Y 445.407,Z 677.096,A -85,B 0,C 180,E1 -8535.377,E2 -8535.377} C_VEL
LIN {X 0,Y 445.339,Z 679.481,A -85,B 0,C 180,E1 -8537.236,E2 -8537.236} C_VEL
LIN {X 0,Y 445.393,Z 680.221,A -85,B 0,C 180,E1 -8538.163,E2 -8538.163} C_VEL
LIN {X 0,Y 445.276,Z 680.824,A -85,B 0,C 180,E1 -8540.002,E2 -8540.002} C_VEL
LIN {X 0,Y 445.325,Z 680.22,A -85,B 0,C 180,E1 -8541.834,E2 -8541.834} C_VEL
LIN {X 0,Y 445.493,Z 678.467,A -85,B 0,C 180,E1 -8543.66,E2 -8543.66} C_VEL
LIN {X 0,Y 445.471,Z 675.562,A -85,B 0,C 180,E1 -8545.476,E2 -8545.476} C_VEL
LIN {X 0,Y 445.681,Z 671.431,A -85,B 0,C 180,E1 -8547.289,E2 -8547.289} C_VEL
LIN {X 0,Y 445.839,Z 666.01,A -85,B 0,C 180,E1 -8549.097,E2 -8549.097} C_VEL
LIN {X 0,Y 446.38,Z 659.118,A -85,B 0,C 180,E1 -8550.902,E2 -8550.902} C_VEL
LIN {X 0,Y 446.99,Z 650.572,A -85,B 0,C 180,E1 -8552.704,E2 -8552.704} C_VEL
LIN {X 0,Y 447.721,Z 641.517,A -85,B 0,C 180,E1 -8554.276,E2 -8554.276} C_VEL
LIN {X 0,Y 448.454,Z 632.341,A -85,B 0,C 180,E1 -8555.621,E2 -8555.621} C_VEL
LIN {X 0,Y 449.475,Z 620.479,A -85,B 0,C 180,E1 -8557.073,E2 -8557.073} C_VEL
LIN {X 0,Y 450.407,Z 608.422,A -85,B 0,C 180,E1 -8558.299,E2 -8558.299} C_VEL
LIN {X 0,Y 451.347,Z 595.199,A -85,B 0,C 180,E1 -8559.41,E2 -8559.41} C_VEL
LIN {X 0,Y 452.298,Z 582.197,A -85,B 0,C 180,E1 -8560.294,E2 -8560.294} C_VEL
LIN {X 0,Y 453.017,Z 569.138,A -85,B 0,C 180,E1 -8561.012,E2 -8561.012} C_VEL
LIN {X 0,Y 453.657,Z 554.949,A -85,B 0,C 180,E1 -8561.619,E2 -8561.619} C_VEL
LIN {X 0,Y 454.108,Z 539.667,A -85,B 0,C 180,E1 -8562.088,E2 -8562.088} C_VEL
LIN {X 0,Y 454.545,Z 518.705,A -85,B 0,C 180,E1 -8562.473,E2 -8562.473} C_VEL
LIN {X 0,Y 456.143,Z 393.889,A -85,B 0,C 180,E1 -8564.478,E2 -8564.478} C_VEL
LIN {X 0,Y 452.407,Z 379.034,A -85,B 0,C 180,E1 -8564.928,E2 -8564.928} C_VEL
LIN {X 0,Y 449.315,Z 371.069,A -85,B 0,C 180,E1 -8565.254,E2 -8565.254} C_VEL
LIN {X 0,Y 446.482,Z 358.498,A -85,B 0,C 180,E1 -8567.757,E2 -8567.757} C_VEL
LIN {X 0,Y 446.448,Z 358.495,A -85,B 0,C 180,E1 -8570.263,E2 -8570.263} C_VEL
LIN {X 0,Y 446.429,Z 358.501,A -85,B 0,C 180,E1 -8573.177,E2 -8573.177} C_VEL
LIN {X 0,Y 446.438,Z 358.498,A -85,B 0,C 180,E1 -8576.191,E2 -8576.191} C_VEL
LIN {X 0,Y 446.427,Z 358.501,A -85,B 0,C 180,E1 -8579.211,E2 -8579.211} C_VEL
LIN {X 0,Y 446.426,Z 358.493,A -85,B 0,C 180,E1 -8582.361,E2 -8582.361} C_VEL
LIN {X 0,Y 446.417,Z 358.499,A -85,B 0,C 180,E1 -8585.626,E2 -8585.626} C_VEL
LIN {X 0,Y 446.404,Z 358.503,A -85,B 0,C 180,E1 -8589.031,E2 -8589.031} C_VEL
LIN {X 0,Y 446.385,Z 358.503,A -85,B 0,C 180,E1 -8592.269,E2 -8592.269} C_VEL
LIN {X 0,Y 446.453,Z 358.494,A -85,B 0,C 180,E1 -8595.104,E2 -8595.104} C_VEL
LIN {X 0,Y 446.41,Z 358.499,A -85,B 0,C 180,E1 -8598.606,E2 -8598.606} C_VEL
LIN {X 0,Y 446.403,Z 358.503,A -85,B 0,C 180,E1 -8601.923,E2 -8601.923} C_VEL
LIN {X 0,Y 446.425,Z 358.5,A -85,B 0,C 180,E1 -8605.476,E2 -8605.476} C_VEL
LIN {X 0,Y 446.417,Z 358.5,A -85,B 0,C 180,E1 -8608.699,E2 -8608.699} C_VEL
LIN {X 0,Y 446.427,Z 358.484,A -85,B 0,C 180,E1 -8611.836,E2 -8611.836} C_VEL
LIN {X 0,Y 446.423,Z 358.476,A -85,B 0,C 180,E1 -8614.845,E2 -8614.845} C_VEL
LIN {X 0,Y 446.452,Z 358.495,A -85,B 0,C 180,E1 -8618.245,E2 -8618.245} C_VEL
LIN {X 0,Y 446.454,Z 358.492,A -85,B 0,C 180,E1 -8621.649,E2 -8621.649} C_VEL
LIN {X 0,Y 446.51,Z 358.486,A -85,B 0,C 180,E1 -8624.479,E2 -8624.479} C_VEL
LIN {X 0,Y 446.52,Z 358.477,A -85,B 0,C 180,E1 -8628.193,E2 -8628.193} C_VEL
LIN {X 0,Y 446.529,Z 358.483,A -85,B 0,C 180,E1 -8630.944,E2 -8630.944} C_VEL
LIN {X 0,Y 446.61,Z 358.473,A -85,B 0,C 180,E1 -8633.675,E2 -8633.675} C_VEL
LIN {X 0,Y 446.657,Z 358.469,A -85,B 0,C 180,E1 -8637.294,E2 -8637.294} C_VEL
LIN {X 0,Y 446.763,Z 358.453,A -85,B 0,C 180,E1 -8640,E2 -8640} C_VEL
LIN {X 0,Y 446.682,Z 358.46,A -85,B 0,C 180,E1 -8642.705,E2 -8642.705} C_VEL
LIN {X 0,Y 446.61,Z 358.472,A -85,B 0,C 180,E1 -8646.324,E2 -8646.324} C_VEL
LIN {X 0,Y 446.533,Z 358.482,A -85,B 0,C 180,E1 -8649.055,E2 -8649.055} C_VEL
LIN {X 0,Y 446.523,Z 358.48,A -85,B 0,C 180,E1 -8652.729,E2 -8652.729} C_VEL
LIN {X 0,Y 446.455,Z 358.492,A -85,B 0,C 180,E1 -8656.208,E2 -8656.208} C_VEL
LIN {X 0,Y 446.469,Z 358.491,A -85,B 0,C 180,E1 -8659.303,E2 -8659.303} C_VEL
LIN {X 0,Y 446.419,Z 358.495,A -85,B 0,C 180,E1 -8662.199,E2 -8662.199} C_VEL
LIN {X 0,Y 446.433,Z 358.498,A -85,B 0,C 180,E1 -8665.153,E2 -8665.153} C_VEL
LIN {X 0,Y 446.439,Z 358.497,A -85,B 0,C 180,E1 -8668.181,E2 -8668.181} C_VEL
LIN {X 0,Y 446.415,Z 358.502,A -85,B 0,C 180,E1 -8671.3,E2 -8671.3} C_VEL
LIN {X 0,Y 446.426,Z 358.498,A -85,B 0,C 180,E1 -8674.523,E2 -8674.523} C_VEL
LIN {X 0,Y 446.398,Z 358.5,A -85,B 0,C 180,E1 -8678.076,E2 -8678.076} C_VEL
LIN {X 0,Y 446.4,Z 358.504,A -85,B 0,C 180,E1 -8681.394,E2 -8681.394} C_VEL
LIN {X 0,Y 446.421,Z 358.5,A -85,B 0,C 180,E1 -8685.107,E2 -8685.107} C_VEL
LIN {X 0,Y 446.406,Z 358.503,A -85,B 0,C 180,E1 -8688.606,E2 -8688.606} C_VEL
LIN {X 0,Y 446.401,Z 358.505,A -85,B 0,C 180,E1 -8691.923,E2 -8691.923} C_VEL
LIN {X 0,Y 446.422,Z 358.505,A -85,B 0,C 180,E1 -8695.476,E2 -8695.476} C_VEL
LIN {X 0,Y 446.46,Z 358.6,A -85,B 0,C 180,E1 -8698.739,E2 -8698.739} C_VEL
LIN {X 0,Y 449.926,Z 372.987,A -85,B 0,C 180,E1 -8701.271,E2 -8701.271} C_VEL
LIN {X 0,Y 451.517,Z 380.359,A -85,B 0,C 180,E1 -8702.526,E2 -8702.526} C_VEL
LIN {X 0,Y 450.685,Z 395.662,A -85,B 0,C 180,E1 -8704.86,E2 -8704.86} C_VEL
LIN {X 0,Y 455.932,Z 423.266,A -85,B 0,C 180,E1 -8705.607,E2 -8705.607} C_VEL
LIN {X 0,Y 454.249,Z 555.293,A -85,B 0,C 180,E1 -8707.725,E2 -8707.725} C_VEL
LIN {X 0,Y 453.861,Z 570.575,A -85,B 0,C 180,E1 -8708.064,E2 -8708.064} C_VEL
LIN {X 0,Y 453.134,Z 585.984,A -85,B 0,C 180,E1 -8708.586,E2 -8708.586} C_VEL
LIN {X 0,Y 452.3,Z 601.129,A -85,B 0,C 180,E1 -8709.298,E2 -8709.298} C_VEL
LIN {X 0,Y 451.435,Z 614.291,A -85,B 0,C 180,E1 -8710.089,E2 -8710.089} C_VEL
LIN {X 0,Y 450.432,Z 627.957,A -85,B 0,C 180,E1 -8711.11,E2 -8711.11} C_VEL
LIN {X 0,Y 449.459,Z 640.445,A -85,B 0,C 180,E1 -8712.247,E2 -8712.247} C_VEL
LIN {X 0,Y 448.47,Z 652.906,A -85,B 0,C 180,E1 -8713.616,E2 -8713.616} C_VEL
LIN {X 0,Y 447.646,Z 663.3,A -85,B 0,C 180,E1 -8714.986,E2 -8714.986} C_VEL
LIN {X 0,Y 446.976,Z 672.108,A -85,B 0,C 180,E1 -8716.358,E2 -8716.358} C_VEL
LIN {X 0,Y 446.406,Z 680.866,A -85,B 0,C 180,E1 -8717.975,E2 -8717.975} C_VEL
LIN {X 0,Y 445.974,Z 688.01,A -85,B 0,C 180,E1 -8719.559,E2 -8719.559} C_VEL
LIN {X 0,Y 445.673,Z 694.7,A -85,B 0,C 180,E1 -8721.384,E2 -8721.384} C_VEL
LIN {X 0,Y 445.504,Z 699.933,A -85,B 0,C 180,E1 -8723.205,E2 -8723.205} C_VEL
LIN {X 0,Y 445.413,Z 702.951,A -85,B 0,C 180,E1 -8724.568,E2 -8724.568} C_VEL
LIN {X 0,Y 445.36,Z 705.902,A -85,B 0,C 180,E1 -8726.381,E2 -8726.381} C_VEL
LIN {X 0,Y 445.371,Z 707.667,A -85,B 0,C 180,E1 -8728.191,E2 -8728.191} C_VEL
LIN {X 0,Y 445.339,Z 708.273,A -85,B 0,C 180,E1 -8730,E2 -8730} C_VEL
LIN {X 0,Y 445.371,Z 707.682,A -85,B 0,C 180,E1 -8731.809,E2 -8731.809} C_VEL
LIN {X 0,Y 445.358,Z 705.947,A -85,B 0,C 180,E1 -8733.619,E2 -8733.619} C_VEL
LIN {X 0,Y 445.407,Z 703.042,A -85,B 0,C 180,E1 -8735.432,E2 -8735.432} C_VEL
LIN {X 0,Y 445.504,Z 698.9,A -85,B 0,C 180,E1 -8737.25,E2 -8737.25} C_VEL
LIN {X 0,Y 445.716,Z 693.415,A -85,B 0,C 180,E1 -8739.072,E2 -8739.072} C_VEL
LIN {X 0,Y 446.132,Z 686.442,A -85,B 0,C 180,E1 -8740.897,E2 -8740.897} C_VEL
LIN {X 0,Y 446.621,Z 677.778,A -85,B 0,C 180,E1 -8742.727,E2 -8742.727} C_VEL
LIN {X 0,Y 447.357,Z 668.596,A -85,B 0,C 180,E1 -8744.326,E2 -8744.326} C_VEL
LIN {X 0,Y 448.074,Z 659.246,A -85,B 0,C 180,E1 -8745.698,E2 -8745.698} C_VEL
LIN {X 0,Y 449.185,Z 647.221,A -85,B 0,C 180,E1 -8747.177,E2 -8747.177} C_VEL
LIN {X 0,Y 450.17,Z 634.964,A -85,B 0,C 180,E1 -8748.43,E2 -8748.43} C_VEL
LIN {X 0,Y 451.292,Z 621.497,A -85,B 0,C 180,E1 -8749.562,E2 -8749.562} C_VEL
LIN {X 0,Y 452.289,Z 608.292,A -85,B 0,C 180,E1 -8750.464,E2 -8750.464} C_VEL
LIN {X 0,Y 453.217,Z 593.943,A -85,B 0,C 180,E1 -8751.248,E2 -8751.248} C_VEL
LIN {X 0,Y 454.037,Z 578.193,A -85,B 0,C 180,E1 -8751.897,E2 -8751.897} C_VEL
LIN {X 0,Y 454.723,Z 562.31,A -85,B 0,C 180,E1 -8752.341,E2 -8752.341} C_VEL
LIN {X 0,Y 456.776,Z 423.222,A -85,B 0,C 180,E1 -8754.629,E2 -8754.629} C_VEL
LIN {X 0,Y 451.597,Z 397.332,A -85,B 0,C 180,E1 -8755.412,E2 -8755.412} C_VEL
LIN {X 0,Y 451.242,Z 395.333,A -85,B 0,C 180,E1 -8755.487,E2 -8755.487} C_VEL
LIN {X 0,Y 452.08,Z 381.816,A -85,B 0,C 180,E1 -8757.611,E2 -8757.611} C_VEL
LIN {X 0,Y 449.464,Z 369.904,A -85,B 0,C 180,E1 -8759.766,E2 -8759.766} C_VEL
LIN {X 0,Y 446.414,Z 358.505,A -85,B 0,C 180,E1 -8761.987,E2 -8761.987} C_VEL
LIN {X 0,Y 446.423,Z 358.503,A -85,B 0,C 180,E1 -8765.052,E2 -8765.052} C_VEL
LIN {X 0,Y 446.402,Z 358.505,A -85,B 0,C 180,E1 -8768.077,E2 -8768.077} C_VEL
LIN {X 0,Y 446.405,Z 358.498,A -85,B 0,C 180,E1 -8771.394,E2 -8771.394} C_VEL
LIN {X 0,Y 446.448,Z 358.497,A -85,B 0,C 180,E1 -8775.104,E2 -8775.104} C_VEL
LIN {X 0,Y 446.4,Z 358.507,A -85,B 0,C 180,E1 -8778.606,E2 -8778.606} C_VEL
LIN {X 0,Y 446.399,Z 358.504,A -85,B 0,C 180,E1 -8781.924,E2 -8781.924} C_VEL
LIN {X 0,Y 446.428,Z 358.495,A -85,B 0,C 180,E1 -8785.477,E2 -8785.477} C_VEL
LIN {X 0,Y 446.415,Z 358.486,A -85,B 0,C 180,E1 -8788.7,E2 -8788.7} C_VEL
LIN {X 0,Y 446.448,Z 358.495,A -85,B 0,C 180,E1 -8791.831,E2 -8791.831} C_VEL
LIN {X 0,Y 446.438,Z 358.499,A -85,B 0,C 180,E1 -8794.847,E2 -8794.847} C_VEL
LIN {X 0,Y 446.449,Z 358.498,A -85,B 0,C 180,E1 -8798.245,E2 -8798.245} C_VEL
LIN {X 0,Y 446.448,Z 358.494,A -85,B 0,C 180,E1 -8801.649,E2 -8801.649} C_VEL
LIN {X 0,Y 446.494,Z 358.491,A -85,B 0,C 180,E1 -8804.48,E2 -8804.48} C_VEL
LIN {X 0,Y 446.518,Z 358.486,A -85,B 0,C 180,E1 -8808.193,E2 -8808.193} C_VEL
LIN {X 0,Y 446.532,Z 358.482,A -85,B 0,C 180,E1 -8810.945,E2 -8810.945} C_VEL
LIN {X 0,Y 446.614,Z 358.475,A -85,B 0,C 180,E1 -8813.676,E2 -8813.676} C_VEL
LIN {X 0,Y 446.683,Z 358.466,A -85,B 0,C 180,E1 -8817.295,E2 -8817.295} C_VEL
LIN {X 0,Y 446.763,Z 358.453,A -85,B 0,C 180,E1 -8820,E2 -8820} C_VEL
LIN {X 0,Y 446.678,Z 358.466,A -85,B 0,C 180,E1 -8822.706,E2 -8822.706} C_VEL
LIN {X 0,Y 446.614,Z 358.479,A -85,B 0,C 180,E1 -8826.325,E2 -8826.325} C_VEL
LIN {X 0,Y 446.532,Z 358.486,A -85,B 0,C 180,E1 -8829.056,E2 -8829.056} C_VEL
LIN {X 0,Y 446.524,Z 358.49,A -85,B 0,C 180,E1 -8832.73,E2 -8832.73} C_VEL
LIN {X 0,Y 446.498,Z 358.492,A -85,B 0,C 180,E1 -8836.228,E2 -8836.228} C_VEL
LIN {X 0,Y 446.471,Z 358.476,A -85,B 0,C 180,E1 -8839.304,E2 -8839.304} C_VEL
LIN {X 0,Y 446.421,Z 358.5,A -85,B 0,C 180,E1 -8842.2,E2 -8842.2} C_VEL
LIN {X 0,Y 446.424,Z 358.486,A -85,B 0,C 180,E1 -8845.155,E2 -8845.155} C_VEL
LIN {X 0,Y 446.443,Z 358.498,A -85,B 0,C 180,E1 -8848.182,E2 -8848.182} C_VEL
LIN {X 0,Y 446.418,Z 358.491,A -85,B 0,C 180,E1 -8851.301,E2 -8851.301} C_VEL
LIN {X 0,Y 446.425,Z 358.496,A -85,B 0,C 180,E1 -8854.524,E2 -8854.524} C_VEL
LIN {X 0,Y 446.403,Z 358.505,A -85,B 0,C 180,E1 -8858.077,E2 -8858.077} C_VEL
LIN {X 0,Y 446.409,Z 358.501,A -85,B 0,C 180,E1 -8861.394,E2 -8861.394} C_VEL
LIN {X 0,Y 446.454,Z 358.493,A -85,B 0,C 180,E1 -8865.104,E2 -8865.104} C_VEL
LIN {X 0,Y 446.422,Z 358.504,A -85,B 0,C 180,E1 -8868.608,E2 -8868.608} C_VEL
LIN {X 0,Y 446.443,Z 358.648,A -85,B 0,C 180,E1 -8871.781,E2 -8871.781} C_VEL
LIN {X 0,Y 449.671,Z 371.711,A -85,B 0,C 180,E1 -8874.479,E2 -8874.479} C_VEL
LIN {X 0,Y 454.481,Z 383.025,A -85,B 0,C 180,E1 -8874.999,E2 -8874.999} C_VEL
LIN {X 0,Y 457.118,Z 394.599,A -85,B 0,C 180,E1 -8875.371,E2 -8875.371} C_VEL
LIN {X 0,Y 455.009,Z 526.107,A -85,B 0,C 180,E1 -8877.505,E2 -8877.505} C_VEL
LIN {X 0,Y 454.813,Z 541.586,A -85,B 0,C 180,E1 -8877.833,E2 -8877.833} C_VEL
LIN {X 0,Y 454.225,Z 555.624,A -85,B 0,C 180,E1 -8878.276,E2 -8878.276} C_VEL
LIN {X 0,Y 453.415,Z 570.929,A -85,B 0,C 180,E1 -8878.95,E2 -8878.95} C_VEL
LIN {X 0,Y 452.619,Z 583.872,A -85,B 0,C 180,E1 -8879.692,E2 -8879.692} C_VEL
LIN {X 0,Y 451.751,Z 596.683,A -85,B 0,C 180,E1 -8880.6,E2 -8880.6} C_VEL
LIN {X 0,Y 451.029,Z 605.377,A -85,B 0,C 180,E1 -8881.327,E2 -8881.327} C_VEL
LIN {X 0,Y 449.999,Z 610.231,A -85,B 0,C 180,E1 -8881.741,E2 -8881.741} C_VEL
LIN {X 0,Y 446.581,Z 617.968,A -85,B 0,C 180,E1 -8882.4,E2 -8882.4} C_VEL
LIN {X 0,Y 443.163,Z 625.407,A -85,B 0,C 180,E1 -8883.123,E2 -8883.123} C_VEL
LIN {X 0,Y 442.147,Z 629.634,A -85,B 0,C 180,E1 -8883.634,E2 -8883.634} C_VEL
LIN {X 0,Y 441.243,Z 639.042,A -85,B 0,C 180,E1 -8884.972,E2 -8884.972} C_VEL
LIN {X 0,Y 440.424,Z 648.062,A -85,B 0,C 180,E1 -8886.488,E2 -8886.488} C_VEL
LIN {X 0,Y 439.762,Z 655.952,A -85,B 0,C 180,E1 -8888.072,E2 -8888.072} C_VEL
LIN {X 0,Y 439.116,Z 663.351,A -85,B 0,C 180,E1 -8889.873,E2 -8889.873} C_VEL
LIN {X 0,Y 438.758,Z 669.646,A -85,B 0,C 180,E1 -8891.799,E2 -8891.799} C_VEL
LIN {X 0,Y 438.53,Z 673.336,A -85,B 0,C 180,E1 -8893.233,E2 -8893.233} C_VEL
LIN {X 0,Y 438.357,Z 677.094,A -85,B 0,C 180,E1 -8895.136,E2 -8895.136} C_VEL
LIN {X 0,Y 438.261,Z 679.579,A -85,B 0,C 180,E1 -8897.026,E2 -8897.026} C_VEL
LIN {X 0,Y 438.323,Z 680.372,A -85,B 0,C 180,E1 -8897.98,E2 -8897.98} C_VEL
LIN {X 0,Y 438.207,Z 681.023,A -85,B 0,C 180,E1 -8899.839,E2 -8899.839} C_VEL
LIN {X 0,Y 438.239,Z 680.512,A -85,B 0,C 180,E1 -8901.701,E2 -8901.701} C_VEL
LIN {X 0,Y 438.407,Z 678.708,A -85,B 0,C 180,E1 -8903.678,E2 -8903.678} C_VEL
LIN {X 0,Y 438.386,Z 676.049,A -85,B 0,C 180,E1 -8905.402,E2 -8905.402} C_VEL
LIN {X 0,Y 438.597,Z 672.019,A -85,B 0,C 180,E1 -8907.245,E2 -8907.245} C_VEL
LIN {X 0,Y 438.759,Z 666.704,A -85,B 0,C 180,E1 -8909.082,E2 -8909.082} C_VEL
LIN {X 0,Y 439.31,Z 659.925,A -85,B 0,C 180,E1 -8910.917,E2 -8910.917} C_VEL
LIN {X 0,Y 439.94,Z 651.508,A -85,B 0,C 180,E1 -8912.747,E2 -8912.747} C_VEL
LIN {X 0,Y 440.713,Z 642.585,A -85,B 0,C 180,E1 -8914.344,E2 -8914.344} C_VEL
LIN {X 0,Y 441.624,Z 631.862,A -85,B 0,C 180,E1 -8915.937,E2 -8915.937} C_VEL
LIN {X 0,Y 442.599,Z 620.86,A -85,B 0,C 180,E1 -8917.298,E2 -8917.298} C_VEL
LIN {X 0,Y 443.567,Z 608.823,A -85,B 0,C 180,E1 -8918.542,E2 -8918.542} C_VEL
LIN {X 0,Y 444.564,Z 595.628,A -85,B 0,C 180,E1 -8919.67,E2 -8919.67} C_VEL
LIN {X 0,Y 445.562,Z 582.658,A -85,B 0,C 180,E1 -8920.566,E2 -8920.566} C_VEL
LIN {X 0,Y 446.309,Z 569.66,A -85,B 0,C 180,E1 -8921.295,E2 -8921.295} C_VEL
LIN {X 0,Y 447.016,Z 554.822,A -85,B 0,C 180,E1 -8921.937,E2 -8921.937} C_VEL
LIN {X 0,Y 447.486,Z 539.363,A -85,B 0,C 180,E1 -8922.414,E2 -8922.414} C_VEL
LIN {X 0,Y 447.921,Z 517.189,A -85,B 0,C 180,E1 -8922.82,E2 -8922.82} C_VEL
LIN {X 0,Y 449.572,Z 394.878,A -85,B 0,C 180,E1 -8924.812,E2 -8924.812} C_VEL
LIN {X 0,Y 446.309,Z 381.903,A -85,B 0,C 180,E1 -8925.212,E2 -8925.212} C_VEL
LIN {X 0,Y 442.171,Z 371.338,A -85,B 0,C 180,E1 -8925.641,E2 -8925.641} C_VEL
LIN {X 0,Y 439.443,Z 359.374,A -85,B 0,C 180,E1 -8928.051,E2 -8928.051} C_VEL
LIN {X 0,Y 439.392,Z 359.371,A -85,B 0,C 180,E1 -8930.603,E2 -8930.603} C_VEL
LIN {X 0,Y 439.375,Z 359.382,A -85,B 0,C 180,E1 -8933.571,E2 -8933.571} C_VEL
LIN {X 0,Y 439.37,Z 359.377,A -85,B 0,C 180,E1 -8936.608,E2 -8936.608} C_VEL
LIN {X 0,Y 439.376,Z 359.378,A -85,B 0,C 180,E1 -8939.727,E2 -8939.727} C_VEL
LIN {X 0,Y 439.377,Z 359.372,A -85,B 0,C 180,E1 -8942.946,E2 -8942.946} C_VEL
LIN {X 0,Y 439.371,Z 359.372,A -85,B 0,C 180,E1 -8946.288,E2 -8946.288} C_VEL
LIN {X 0,Y 439.362,Z 359.375,A -85,B 0,C 180,E1 -8949.78,E2 -8949.78} C_VEL
LIN {X 0,Y 439.336,Z 359.38,A -85,B 0,C 180,E1 -8952.62,E2 -8952.62} C_VEL
LIN {X 0,Y 439.401,Z 359.371,A -85,B 0,C 180,E1 -8955.27,E2 -8955.27} C_VEL
LIN {X 0,Y 439.36,Z 359.379,A -85,B 0,C 180,E1 -8959.016,E2 -8959.016} C_VEL
LIN {X 0,Y 439.341,Z 359.38,A -85,B 0,C 180,E1 -8962.563,E2 -8962.563} C_VEL
LIN {X 0,Y 439.398,Z 359.373,A -85,B 0,C 180,E1 -8964.843,E2 -8964.843} C_VEL
LIN {X 0,Y 439.373,Z 359.379,A -85,B 0,C 180,E1 -8968.139,E2 -8968.139} C_VEL
LIN {X 0,Y 439.403,Z 359.362,A -85,B 0,C 180,E1 -8971.606,E2 -8971.606} C_VEL
LIN {X 0,Y 439.368,Z 359.354,A -85,B 0,C 180,E1 -8974.412,E2 -8974.412} C_VEL
LIN {X 0,Y 439.367,Z 359.375,A -85,B 0,C 180,E1 -8977.424,E2 -8977.424} C_VEL
LIN {X 0,Y 439.444,Z 359.366,A -85,B 0,C 180,E1 -8980.663,E2 -8980.663} C_VEL
LIN {X 0,Y 439.465,Z 359.364,A -85,B 0,C 180,E1 -8984.224,E2 -8984.224} C_VEL
LIN {X 0,Y 439.486,Z 359.354,A -85,B 0,C 180,E1 -8988.001,E2 -8988.001} C_VEL
LIN {X 0,Y 439.504,Z 359.364,A -85,B 0,C 180,E1 -8991.725,E2 -8991.725} C_VEL
LIN {X 0,Y 439.601,Z 359.339,A -85,B 0,C 180,E1 -8994.495,E2 -8994.495} C_VEL
LIN {X 0,Y 439.629,Z 359.345,A -85,B 0,C 180,E1 -8998.167,E2 -8998.167} C_VEL
LIN {X 0,Y 439.712,Z 359.331,A -85,B 0,C 180,E1 -9000,E2 -9000} C_VEL
LIN {X 0,Y 439.631,Z 359.339,A -85,B 0,C 180,E1 -9002.748,E2 -9002.748} C_VEL
LIN {X 0,Y 439.563,Z 359.35,A -85,B 0,C 180,E1 -9006.426,E2 -9006.426} C_VEL
LIN {X 0,Y 439.496,Z 359.359,A -85,B 0,C 180,E1 -9009.201,E2 -9009.201} C_VEL
LIN {X 0,Y 439.467,Z 359.359,A -85,B 0,C 180,E1 -9012.937,E2 -9012.937} C_VEL
LIN {X 0,Y 439.404,Z 359.37,A -85,B 0,C 180,E1 -9016.328,E2 -9016.328} C_VEL
LIN {X 0,Y 439.403,Z 359.376,A -85,B 0,C 180,E1 -9019.626,E2 -9019.626} C_VEL
LIN {X 0,Y 439.364,Z 359.372,A -85,B 0,C 180,E1 -9022.575,E2 -9022.575} C_VEL
LIN {X 0,Y 439.373,Z 359.379,A -85,B 0,C 180,E1 -9025.587,E2 -9025.587} C_VEL
LIN {X 0,Y 439.392,Z 359.374,A -85,B 0,C 180,E1 -9028.675,E2 -9028.675} C_VEL
LIN {X 0,Y 439.37,Z 359.378,A -85,B 0,C 180,E1 -9032.03,E2 -9032.03} C_VEL
LIN {X 0,Y 439.39,Z 359.378,A -85,B 0,C 180,E1 -9035.339,E2 -9035.339} C_VEL
LIN {X 0,Y 439.354,Z 359.375,A -85,B 0,C 180,E1 -9038.598,E2 -9038.598} C_VEL
LIN {X 0,Y 439.348,Z 359.38,A -85,B 0,C 180,E1 -9042.21,E2 -9042.21} C_VEL
LIN {X 0,Y 439.375,Z 359.38,A -85,B 0,C 180,E1 -9045.267,E2 -9045.267} C_VEL
LIN {X 0,Y 439.367,Z 359.38,A -85,B 0,C 180,E1 -9048.746,E2 -9048.746} C_VEL
LIN {X 0,Y 439.358,Z 359.384,A -85,B 0,C 180,E1 -9051.61,E2 -9051.61} C_VEL
LIN {X 0,Y 439.394,Z 359.376,A -85,B 0,C 180,E1 -9054.843,E2 -9054.843} C_VEL
LIN {X 0,Y 439.371,Z 359.38,A -85,B 0,C 180,E1 -9058.139,E2 -9058.139} C_VEL
LIN {X 0,Y 439.391,Z 359.459,A -85,B 0,C 180,E1 -9058.41,E2 -9058.41} C_VEL
LIN {X 0,Y 443.139,Z 374.985,A -85,B 0,C 180,E1 -9061.19,E2 -9061.19} C_VEL
LIN {X 0,Y 444.692,Z 382.428,A -85,B 0,C 180,E1 -9062.471,E2 -9062.471} C_VEL
LIN {X 0,Y 443.899,Z 395.412,A -85,B 0,C 180,E1 -9064.481,E2 -9064.481} C_VEL
LIN {X 0,Y 449.423,Z 424.992,A -85,B 0,C 180,E1 -9065.295,E2 -9065.295} C_VEL
LIN {X 0,Y 447.463,Z 561.071,A -85,B 0,C 180,E1 -9067.52,E2 -9067.52} C_VEL
LIN {X 0,Y 446.871,Z 576.743,A -85,B 0,C 180,E1 -9067.945,E2 -9067.945} C_VEL
LIN {X 0,Y 446.096,Z 592.083,A -85,B 0,C 180,E1 -9068.554,E2 -9068.554} C_VEL
LIN {X 0,Y 445.191,Z 606.427,A -85,B 0,C 180,E1 -9069.315,E2 -9069.315} C_VEL
LIN {X 0,Y 444.23,Z 620.094,A -85,B 0,C 180,E1 -9070.235,E2 -9070.235} C_VEL
LIN {X 0,Y 443.07,Z 633.967,A -85,B 0,C 180,E1 -9071.384,E2 -9071.384} C_VEL
LIN {X 0,Y 442.001,Z 646.748,A -85,B 0,C 180,E1 -9072.682,E2 -9072.682} C_VEL
LIN {X 0,Y 441.087,Z 657.908,A -85,B 0,C 180,E1 -9074.047,E2 -9074.047} C_VEL
LIN {X 0,Y 440.252,Z 668.996,A -85,B 0,C 180,E1 -9075.674,E2 -9075.674} C_VEL
LIN {X 0,Y 439.452,Z 678.912,A -85,B 0,C 180,E1 -9077.446,E2 -9077.446} C_VEL
LIN {X 0,Y 439.102,Z 685.782,A -85,B 0,C 180,E1 -9078.927,E2 -9078.927} C_VEL
LIN {X 0,Y 438.65,Z 692.883,A -85,B 0,C 180,E1 -9080.78,E2 -9080.78} C_VEL
LIN {X 0,Y 438.485,Z 698.472,A -85,B 0,C 180,E1 -9082.633,E2 -9082.633} C_VEL
LIN {X 0,Y 438.317,Z 702.694,A -85,B 0,C 180,E1 -9084.479,E2 -9084.479} C_VEL
LIN {X 0,Y 438.26,Z 705.66,A -85,B 0,C 180,E1 -9086.322,E2 -9086.322} C_VEL
LIN {X 0,Y 438.292,Z 707.439,A -85,B 0,C 180,E1 -9088.162,E2 -9088.162} C_VEL
LIN {X 0,Y 438.25,Z 708.053,A -85,B 0,C 180,E1 -9090,E2 -9090} C_VEL
LIN {X 0,Y 438.292,Z 707.473,A -85,B 0,C 180,E1 -9091.838,E2 -9091.838} C_VEL
LIN {X 0,Y 438.259,Z 705.75,A -85,B 0,C 180,E1 -9093.678,E2 -9093.678} C_VEL
LIN {X 0,Y 438.311,Z 702.859,A -85,B 0,C 180,E1 -9095.521,E2 -9095.521} C_VEL
LIN {X 0,Y 438.43,Z 698.734,A -85,B 0,C 180,E1 -9097.368,E2 -9097.368} C_VEL
LIN {X 0,Y 438.649,Z 693.268,A -85,B 0,C 180,E1 -9099.22,E2 -9099.22} C_VEL
LIN {X 0,Y 439.107,Z 686.319,A -85,B 0,C 180,E1 -9101.073,E2 -9101.073} C_VEL
LIN {X 0,Y 439.65,Z 677.684,A -85,B 0,C 180,E1 -9102.932,E2 -9102.932} C_VEL
LIN {X 0,Y 440.424,Z 668.536,A -85,B 0,C 180,E1 -9104.556,E2 -9104.556} C_VEL
LIN {X 0,Y 441.369,Z 657.506,A -85,B 0,C 180,E1 -9106.18,E2 -9106.18} C_VEL
LIN {X 0,Y 442.439,Z 646.206,A -85,B 0,C 180,E1 -9107.566,E2 -9107.566} C_VEL
LIN {X 0,Y 443.506,Z 633.813,A -85,B 0,C 180,E1 -9108.837,E2 -9108.837} C_VEL
LIN {X 0,Y 444.696,Z 620.132,A -85,B 0,C 180,E1 -9109.984,E2 -9109.984} C_VEL
LIN {X 0,Y 445.786,Z 606.738,A -85,B 0,C 180,E1 -9110.897,E2 -9110.897} C_VEL
LIN {X 0,Y 446.747,Z 592.456,A -85,B 0,C 180,E1 -9111.671,E2 -9111.671} C_VEL
LIN {X 0,Y 447.58,Z 577.249,A -85,B 0,C 180,E1 -9112.291,E2 -9112.291} C_VEL
LIN {X 0,Y 448.266,Z 562.188,A -85,B 0,C 180,E1 -9112.711,E2 -9112.711} C_VEL
LIN {X 0,Y 450.467,Z 424.618,A -85,B 0,C 180,E1 -9115.005,E2 -9115.005} C_VEL
LIN {X 0,Y 445.56,Z 399.71,A -85,B 0,C 180,E1 -9115.772,E2 -9115.772} C_VEL
LIN {X 0,Y 444.605,Z 395.099,A -85,B 0,C 180,E1 -9115.937,E2 -9115.937} C_VEL
LIN {X 0,Y 445.369,Z 384.248,A -85,B 0,C 180,E1 -9117.668,E2 -9117.668} C_VEL
LIN {X 0,Y 443.412,Z 374.584,A -85,B 0,C 180,E1 -9119.429,E2 -9119.429} C_VEL
LIN {X 0,Y 440.142,Z 362.363,A -85,B 0,C 180,E1 -9121.798,E2 -9121.798} C_VEL
LIN {X 0,Y 439.391,Z 359.381,A -85,B 0,C 180,E1 -9122.413,E2 -9122.413} C_VEL
LIN {X 0,Y 439.389,Z 359.379,A -85,B 0,C 180,E1 -9125.34,E2 -9125.34} C_VEL
LIN {X 0,Y 439.355,Z 359.377,A -85,B 0,C 180,E1 -9128.598,E2 -9128.598} C_VEL
LIN {X 0,Y 439.357,Z 359.375,A -85,B 0,C 180,E1 -9132.209,E2 -9132.209} C_VEL
LIN {X 0,Y 439.396,Z 359.375,A -85,B 0,C 180,E1 -9135.27,E2 -9135.27} C_VEL
LIN {X 0,Y 439.353,Z 359.381,A -85,B 0,C 180,E1 -9139.016,E2 -9139.016} C_VEL
LIN {X 0,Y 439.336,Z 359.377,A -85,B 0,C 180,E1 -9142.564,E2 -9142.564} C_VEL
LIN {X 0,Y 439.397,Z 359.371,A -85,B 0,C 180,E1 -9144.844,E2 -9144.844} C_VEL
LIN {X 0,Y 439.372,Z 359.37,A -85,B 0,C 180,E1 -9148.14,E2 -9148.14} C_VEL
LIN {X 0,Y 439.403,Z 359.372,A -85,B 0,C 180,E1 -9151.606,E2 -9151.606} C_VEL
LIN {X 0,Y 439.377,Z 359.378,A -85,B 0,C 180,E1 -9154.414,E2 -9154.414} C_VEL
LIN {X 0,Y 439.363,Z 359.375,A -85,B 0,C 180,E1 -9157.425,E2 -9157.425} C_VEL
LIN {X 0,Y 439.441,Z 359.369,A -85,B 0,C 180,E1 -9160.664,E2 -9160.664} C_VEL
LIN {X 0,Y 439.455,Z 359.367,A -85,B 0,C 180,E1 -9164.225,E2 -9164.225} C_VEL
LIN {X 0,Y 439.484,Z 359.361,A -85,B 0,C 180,E1 -9168.002,E2 -9168.002} C_VEL
LIN {X 0,Y 439.504,Z 359.356,A -85,B 0,C 180,E1 -9171.726,E2 -9171.726} C_VEL
LIN {X 0,Y 439.606,Z 359.35,A -85,B 0,C 180,E1 -9174.496,E2 -9174.496} C_VEL
LIN {X 0,Y 439.634,Z 359.348,A -85,B 0,C 180,E1 -9178.168,E2 -9178.168} C_VEL
LIN {X 0,Y 439.712,Z 359.331,A -85,B 0,C 180,E1 -9180,E2 -9180} C_VEL
LIN {X 0,Y 439.628,Z 359.343,A -85,B 0,C 180,E1 -9182.749,E2 -9182.749} C_VEL
LIN {X 0,Y 439.565,Z 359.355,A -85,B 0,C 180,E1 -9186.426,E2 -9186.426} C_VEL
LIN {X 0,Y 439.496,Z 359.362,A -85,B 0,C 180,E1 -9189.202,E2 -9189.202} C_VEL
LIN {X 0,Y 439.468,Z 359.367,A -85,B 0,C 180,E1 -9192.938,E2 -9192.938} C_VEL
LIN {X 0,Y 439.449,Z 359.372,A -85,B 0,C 180,E1 -9196.348,E2 -9196.348} C_VEL
LIN {X 0,Y 439.405,Z 359.355,A -85,B 0,C 180,E1 -9199.627,E2 -9199.627} C_VEL
LIN {X 0,Y 439.366,Z 359.384,A -85,B 0,C 180,E1 -9202.576,E2 -9202.576} C_VEL
LIN {X 0,Y 439.369,Z 359.363,A -85,B 0,C 180,E1 -9205.588,E2 -9205.588} C_VEL
LIN {X 0,Y 439.399,Z 359.378,A -85,B 0,C 180,E1 -9208.675,E2 -9208.675} C_VEL
LIN {X 0,Y 439.372,Z 359.371,A -85,B 0,C 180,E1 -9212.03,E2 -9212.03} C_VEL
LIN {X 0,Y 439.393,Z 359.364,A -85,B 0,C 180,E1 -9215.34,E2 -9215.34} C_VEL
LIN {X 0,Y 439.358,Z 359.377,A -85,B 0,C 180,E1 -9218.598,E2 -9218.598} C_VEL
LIN {X 0,Y 439.361,Z 359.378,A -85,B 0,C 180,E1 -9222.209,E2 -9222.209} C_VEL
LIN {X 0,Y 439.402,Z 359.371,A -85,B 0,C 180,E1 -9225.271,E2 -9225.271} C_VEL
LIN {X 0,Y 439.385,Z 359.382,A -85,B 0,C 180,E1 -9228.745,E2 -9228.745} C_VEL
LIN {X 0,Y 439.373,Z 359.386,A -85,B 0,C 180,E1 -9231.331,E2 -9231.331} C_VEL
LIN {X 0,Y 442.431,Z 371.766,A -85,B 0,C 180,E1 -9233.978,E2 -9233.978} C_VEL
LIN {X 0,Y 448.527,Z 385.761,A -85,B 0,C 180,E1 -9234.652,E2 -9234.652} C_VEL
LIN {X 0,Y 450.785,Z 395.706,A -85,B 0,C 180,E1 -9234.979,E2 -9234.979} C_VEL
LIN {X 0,Y 448.645,Z 523.591,A -85,B 0,C 180,E1 -9237.086,E2 -9237.086} C_VEL
LIN {X 0,Y 448.38,Z 540.619,A -85,B 0,C 180,E1 -9237.431,E2 -9237.431} C_VEL
LIN {X 0,Y 447.71,Z 555.725,A -85,B 0,C 180,E1 -9237.904,E2 -9237.904} C_VEL
LIN {X 0,Y 446.942,Z 570.222,A -85,B 0,C 180,E1 -9238.546,E2 -9238.546} C_VEL
LIN {X 0,Y 446.074,Z 583.848,A -85,B 0,C 180,E1 -9239.331,E2 -9239.331} C_VEL
LIN {X 0,Y 445.102,Z 597.043,A -85,B 0,C 180,E1 -9240.278,E2 -9240.278} C_VEL
LIN {X 0,Y 443.964,Z 609.769,A -85,B 0,C 180,E1 -9241.389,E2 -9241.389} C_VEL
LIN {X 0,Y 442.836,Z 622.26,A -85,B 0,C 180,E1 -9242.717,E2 -9242.717} C_VEL
LIN {X 0,Y 442.147,Z 629.634,A -85,B 0,C 180,E1 -9243.634,E2 -9243.634} C_VEL
LIN {X 0,Y 441.234,Z 632.491,A -85,B 0,C 180,E1 -9243.981,E2 -9243.981} C_VEL
LIN {X 0,Y 434.833,Z 641.252,A -85,B 0,C 180,E1 -9245.033,E2 -9245.033} C_VEL
LIN {X 0,Y 433.964,Z 643.735,A -85,B 0,C 180,E1 -9245.426,E2 -9245.426} C_VEL
LIN {X 0,Y 433.072,Z 652.593,A -85,B 0,C 180,E1 -9247.078,E2 -9247.078} C_VEL
LIN {X 0,Y 432.528,Z 659.196,A -85,B 0,C 180,E1 -9248.556,E2 -9248.556} C_VEL
LIN {X 0,Y 431.929,Z 666.139,A -85,B 0,C 180,E1 -9250.426,E2 -9250.426} C_VEL
LIN {X 0,Y 431.552,Z 672.06,A -85,B 0,C 180,E1 -9252.466,E2 -9252.466} C_VEL
LIN {X 0,Y 431.405,Z 675.447,A -85,B 0,C 180,E1 -9253.982,E2 -9253.982} C_VEL
LIN {X 0,Y 431.186,Z 678.543,A -85,B 0,C 180,E1 -9255.848,E2 -9255.848} C_VEL
LIN {X 0,Y 431.223,Z 680.596,A -85,B 0,C 180,E1 -9257.926,E2 -9257.926} C_VEL
LIN {X 0,Y 431.113,Z 681.219,A -85,B 0,C 180,E1 -9259.67,E2 -9259.67} C_VEL
LIN {X 0,Y 431.134,Z 680.802,A -85,B 0,C 180,E1 -9261.564,E2 -9261.564} C_VEL
LIN {X 0,Y 431.31,Z 678.931,A -85,B 0,C 180,E1 -9263.709,E2 -9263.709} C_VEL
LIN {X 0,Y 431.304,Z 676.529,A -85,B 0,C 180,E1 -9265.327,E2 -9265.327} C_VEL
LIN {X 0,Y 431.516,Z 672.594,A -85,B 0,C 180,E1 -9267.199,E2 -9267.199} C_VEL
LIN {X 0,Y 431.675,Z 667.354,A -85,B 0,C 180,E1 -9269.067,E2 -9269.067} C_VEL
LIN {X 0,Y 432.236,Z 660.676,A -85,B 0,C 180,E1 -9270.932,E2 -9270.932} C_VEL
LIN {X 0,Y 432.894,Z 652.401,A -85,B 0,C 180,E1 -9272.792,E2 -9272.792} C_VEL
LIN {X 0,Y 433.684,Z 643.581,A -85,B 0,C 180,E1 -9274.415,E2 -9274.415} C_VEL
LIN {X 0,Y 434.627,Z 633.026,A -85,B 0,C 180,E1 -9276.033,E2 -9276.033} C_VEL
LIN {X 0,Y 435.632,Z 622.176,A -85,B 0,C 180,E1 -9277.416,E2 -9277.416} C_VEL
LIN {X 0,Y 436.655,Z 610.342,A -85,B 0,C 180,E1 -9278.679,E2 -9278.679} C_VEL
LIN {X 0,Y 437.705,Z 597.411,A -85,B 0,C 180,E1 -9279.823,E2 -9279.823} C_VEL
LIN {X 0,Y 438.68,Z 584.824,A -85,B 0,C 180,E1 -9280.734,E2 -9280.734} C_VEL
LIN {X 0,Y 439.516,Z 571.253,A -85,B 0,C 180,E1 -9281.53,E2 -9281.53} C_VEL
LIN {X 0,Y 440.3,Z 556.129,A -85,B 0,C 180,E1 -9282.21,E2 -9282.21} C_VEL
LIN {X 0,Y 440.836,Z 540.086,A -85,B 0,C 180,E1 -9282.721,E2 -9282.721} C_VEL
LIN {X 0,Y 441.295,Z 519.105,A -85,B 0,C 180,E1 -9283.117,E2 -9283.117} C_VEL
LIN {X 0,Y 443.056,Z 396.272,A -85,B 0,C 180,E1 -9285.143,E2 -9285.143} C_VEL
LIN {X 0,Y 439.974,Z 384.161,A -85,B 0,C 180,E1 -9285.526,E2 -9285.526} C_VEL
LIN {X 0,Y 434.98,Z 371.497,A -85,B 0,C 180,E1 -9286.062,E2 -9286.062} C_VEL
LIN {X 0,Y 432.396,Z 360.252,A -85,B 0,C 180,E1 -9288.356,E2 -9288.356} C_VEL
LIN {X 0,Y 432.363,Z 360.255,A -85,B 0,C 180,E1 -9291.954,E2 -9291.954} C_VEL
LIN {X 0,Y 432.328,Z 360.256,A -85,B 0,C 180,E1 -9295.003,E2 -9295.003} C_VEL
LIN {X 0,Y 432.351,Z 360.252,A -85,B 0,C 180,E1 -9298.622,E2 -9298.622} C_VEL
LIN {X 0,Y 432.325,Z 360.259,A -85,B 0,C 180,E1 -9301.346,E2 -9301.346} C_VEL
LIN {X 0,Y 432.341,Z 360.253,A -85,B 0,C 180,E1 -9304.677,E2 -9304.677} C_VEL
LIN {X 0,Y 432.326,Z 360.256,A -85,B 0,C 180,E1 -9308.151,E2 -9308.151} C_VEL
LIN {X 0,Y 432.307,Z 360.259,A -85,B 0,C 180,E1 -9311.8,E2 -9311.8} C_VEL
LIN {X 0,Y 432.337,Z 360.25,A -85,B 0,C 180,E1 -9314.347,E2 -9314.347} C_VEL
LIN {X 0,Y 432.31,Z 360.249,A -85,B 0,C 180,E1 -9317.017,E2 -9317.017} C_VEL
LIN {X 0,Y 432.292,Z 360.26,A -85,B 0,C 180,E1 -9319.828,E2 -9319.828} C_VEL
LIN {X 0,Y 432.302,Z 360.258,A -85,B 0,C 180,E1 -9323.021,E2 -9323.021} C_VEL
LIN {X 0,Y 432.336,Z 360.253,A -85,B 0,C 180,E1 -9326.002,E2 -9326.002} C_VEL
LIN {X 0,Y 432.35,Z 360.257,A -85,B 0,C 180,E1 -9329.49,E2 -9329.49} C_VEL
LIN {X 0,Y 432.331,Z 360.238,A -85,B 0,C 180,E1 -9331.872,E2 -9331.872} C_VEL
LIN {X 0,Y 432.356,Z 360.234,A -85,B 0,C 180,E1 -9335.546,E2 -9335.546} C_VEL
LIN {X 0,Y 432.354,Z 360.252,A -85,B 0,C 180,E1 -9339.046,E2 -9339.046} C_VEL
LIN {X 0,Y 432.363,Z 360.243,A -85,B 0,C 180,E1 -9342.01,E2 -9342.01} C_VEL
LIN {X 0,Y 432.396,Z 360.245,A -85,B 0,C 180,E1 -9344.926,E2 -9344.926} C_VEL
LIN {X 0,Y 432.462,Z 360.231,A -85,B 0,C 180,E1 -9347.803,E2 -9347.803} C_VEL
LIN {X 0,Y 432.465,Z 360.242,A -85,B 0,C 180,E1 -9351.589,E2 -9351.589} C_VEL
LIN {X 0,Y 432.556,Z 360.216,A -85,B 0,C 180,E1 -9354.405,E2 -9354.405} C_VEL
LIN {X 0,Y 432.598,Z 360.221,A -85,B 0,C 180,E1 -9358.138,E2 -9358.138} C_VEL
LIN {X 0,Y 432.662,Z 360.209,A -85,B 0,C 180,E1 -9360,E2 -9360} C_VEL
LIN {X 0,Y 432.583,Z 360.217,A -85,B 0,C 180,E1 -9362.793,E2 -9362.793} C_VEL
LIN {X 0,Y 432.575,Z 360.228,A -85,B 0,C 180,E1 -9365.594,E2 -9365.594} C_VEL
LIN {X 0,Y 432.465,Z 360.232,A -85,B 0,C 180,E1 -9368.41,E2 -9368.41} C_VEL
LIN {X 0,Y 432.461,Z 360.232,A -85,B 0,C 180,E1 -9372.196,E2 -9372.196} C_VEL
LIN {X 0,Y 432.39,Z 360.245,A -85,B 0,C 180,E1 -9376.04,E2 -9376.04} C_VEL
LIN {X 0,Y 432.388,Z 360.247,A -85,B 0,C 180,E1 -9379.484,E2 -9379.484} C_VEL
LIN {X 0,Y 432.318,Z 360.251,A -85,B 0,C 180,E1 -9382.964,E2 -9382.964} C_VEL
LIN {X 0,Y 432.335,Z 360.253,A -85,B 0,C 180,E1 -9385.002,E2 -9385.002} C_VEL
LIN {X 0,Y 432.348,Z 360.251,A -85,B 0,C 180,E1 -9388.622,E2 -9388.622} C_VEL
LIN {X 0,Y 432.321,Z 360.258,A -85,B 0,C 180,E1 -9391.346,E2 -9391.346} C_VEL
LIN {X 0,Y 432.337,Z 360.253,A -85,B 0,C 180,E1 -9394.677,E2 -9394.677} C_VEL
LIN {X 0,Y 432.321,Z 360.253,A -85,B 0,C 180,E1 -9398.151,E2 -9398.151} C_VEL
LIN {X 0,Y 432.303,Z 360.262,A -85,B 0,C 180,E1 -9401.8,E2 -9401.8} C_VEL
LIN {X 0,Y 432.331,Z 360.255,A -85,B 0,C 180,E1 -9404.347,E2 -9404.347} C_VEL
LIN {X 0,Y 432.306,Z 360.26,A -85,B 0,C 180,E1 -9407.017,E2 -9407.017} C_VEL
LIN {X 0,Y 432.288,Z 360.263,A -85,B 0,C 180,E1 -9409.828,E2 -9409.828} C_VEL
LIN {X 0,Y 432.298,Z 360.262,A -85,B 0,C 180,E1 -9413.021,E2 -9413.021} C_VEL
LIN {X 0,Y 432.357,Z 360.256,A -85,B 0,C 180,E1 -9415.997,E2 -9415.997} C_VEL
LIN {X 0,Y 432.369,Z 360.383,A -85,B 0,C 180,E1 -9418.086,E2 -9418.086} C_VEL
LIN {X 0,Y 435.973,Z 375.18,A -85,B 0,C 180,E1 -9420.789,E2 -9420.789} C_VEL
LIN {X 0,Y 437.801,Z 383.502,A -85,B 0,C 180,E1 -9422.255,E2 -9422.255} C_VEL
LIN {X 0,Y 437.159,Z 395.187,A -85,B 0,C 180,E1 -9424.097,E2 -9424.097} C_VEL
LIN {X 0,Y 442.844,Z 426.278,A -85,B 0,C 180,E1 -9424.967,E2 -9424.967} C_VEL
LIN {X 0,Y 440.802,Z 562.082,A -85,B 0,C 180,E1 -9427.224,E2 -9427.224} C_VEL
LIN {X 0,Y 440.154,Z 577.871,A -85,B 0,C 180,E1 -9427.674,E2 -9427.674} C_VEL
LIN {X 0,Y 439.391,Z 591.934,A -85,B 0,C 180,E1 -9428.248,E2 -9428.248} C_VEL
LIN {X 0,Y 438.494,Z 605.665,A -85,B 0,C 180,E1 -9428.985,E2 -9428.985} C_VEL
LIN {X 0,Y 437.47,Z 619.449,A -85,B 0,C 180,E1 -9429.916,E2 -9429.916} C_VEL
LIN {X 0,Y 436.284,Z 633.408,A -85,B 0,C 180,E1 -9431.083,E2 -9431.083} C_VEL
LIN {X 0,Y 435.27,Z 645.266,A -85,B 0,C 180,E1 -9432.294,E2 -9432.294} C_VEL
LIN {X 0,Y 434.38,Z 655.666,A -85,B 0,C 180,E1 -9433.552,E2 -9433.552} C_VEL
LIN {X 0,Y 433.491,Z 665.594,A -85,B 0,C 180,E1 -9434.965,E2 -9434.965} C_VEL
LIN {X 0,Y 432.664,Z 675.311,A -85,B 0,C 180,E1 -9436.616,E2 -9436.616} C_VEL
LIN {X 0,Y 432.131,Z 683.405,A -85,B 0,C 180,E1 -9438.27,E2 -9438.27} C_VEL
LIN {X 0,Y 431.656,Z 690.944,A -85,B 0,C 180,E1 -9440.157,E2 -9440.157} C_VEL
LIN {X 0,Y 431.41,Z 696.929,A -85,B 0,C 180,E1 -9442.041,E2 -9442.041} C_VEL
LIN {X 0,Y 431.256,Z 701.199,A -85,B 0,C 180,E1 -9443.767,E2 -9443.767} C_VEL
LIN {X 0,Y 431.218,Z 704.075,A -85,B 0,C 180,E1 -9445.326,E2 -9445.326} C_VEL
LIN {X 0,Y 431.228,Z 706.458,A -85,B 0,C 180,E1 -9447.197,E2 -9447.197} C_VEL
LIN {X 0,Y 431.168,Z 707.672,A -85,B 0,C 180,E1 -9449.066,E2 -9449.066} C_VEL
LIN {X 0,Y 431.168,Z 707.69,A -85,B 0,C 180,E1 -9450.934,E2 -9450.934} C_VEL
LIN {X 0,Y 431.227,Z 706.557,A -85,B 0,C 180,E1 -9452.802,E2 -9452.802} C_VEL
LIN {X 0,Y 431.216,Z 704.271,A -85,B 0,C 180,E1 -9454.674,E2 -9454.674} C_VEL
LIN {X 0,Y 431.28,Z 700.791,A -85,B 0,C 180,E1 -9456.55,E2 -9456.55} C_VEL
LIN {X 0,Y 431.465,Z 696.032,A -85,B 0,C 180,E1 -9458.43,E2 -9458.43} C_VEL
LIN {X 0,Y 431.746,Z 689.866,A -85,B 0,C 180,E1 -9460.315,E2 -9460.315} C_VEL
LIN {X 0,Y 432.244,Z 683.174,A -85,B 0,C 180,E1 -9461.965,E2 -9461.965} C_VEL
LIN {X 0,Y 432.869,Z 675.139,A -85,B 0,C 180,E1 -9463.616,E2 -9463.616} C_VEL
LIN {X 0,Y 433.731,Z 665.521,A -85,B 0,C 180,E1 -9465.266,E2 -9465.266} C_VEL
LIN {X 0,Y 434.673,Z 655.73,A -85,B 0,C 180,E1 -9466.678,E2 -9466.678} C_VEL
LIN {X 0,Y 435.829,Z 644.13,A -85,B 0,C 180,E1 -9468.084,E2 -9468.084} C_VEL
LIN {X 0,Y 436.893,Z 632.651,A -85,B 0,C 180,E1 -9469.255,E2 -9469.255} C_VEL
LIN {X 0,Y 438.03,Z 620.347,A -85,B 0,C 180,E1 -9470.302,E2 -9470.302} C_VEL
LIN {X 0,Y 439.174,Z 607.038,A -85,B 0,C 180,E1 -9471.227,E2 -9471.227} C_VEL
LIN {X 0,Y 440.266,Z 591.687,A -85,B 0,C 180,E1 -9472.069,E2 -9472.069} C_VEL
LIN {X 0,Y 441.099,Z 577.161,A -85,B 0,C 180,E1 -9472.667,E2 -9472.667} C_VEL
LIN {X 0,Y 441.823,Z 562.165,A -85,B 0,C 180,E1 -9473.092,E2 -9473.092} C_VEL
LIN {X 0,Y 443.915,Z 438.419,A -85,B 0,C 180,E1 -9475.189,E2 -9475.189} C_VEL
LIN {X 0,Y 444.02,Z 425.132,A -85,B 0,C 180,E1 -9475.42,E2 -9475.42} C_VEL
LIN {X 0,Y 439.49,Z 401.982,A -85,B 0,C 180,E1 -9476.151,E2 -9476.151} C_VEL
LIN {X 0,Y 437.926,Z 394.806,A -85,B 0,C 180,E1 -9476.418,E2 -9476.418} C_VEL
LIN {X 0,Y 438.561,Z 385.553,A -85,B 0,C 180,E1 -9477.926,E2 -9477.926} C_VEL
LIN {X 0,Y 435.846,Z 373.257,A -85,B 0,C 180,E1 -9480.239,E2 -9480.239} C_VEL
LIN {X 0,Y 432.352,Z 360.257,A -85,B 0,C 180,E1 -9482.855,E2 -9482.855} C_VEL
LIN {X 0,Y 432.334,Z 360.256,A -85,B 0,C 180,E1 -9485.818,E2 -9485.818} C_VEL
LIN {X 0,Y 432.299,Z 360.255,A -85,B 0,C 180,E1 -9489.348,E2 -9489.348} C_VEL
LIN {X 0,Y 432.307,Z 360.252,A -85,B 0,C 180,E1 -9491.8,E2 -9491.8} C_VEL
LIN {X 0,Y 432.332,Z 360.258,A -85,B 0,C 180,E1 -9494.348,E2 -9494.348} C_VEL
LIN {X 0,Y 432.302,Z 360.26,A -85,B 0,C 180,E1 -9497.018,E2 -9497.018} C_VEL
LIN {X 0,Y 432.287,Z 360.262,A -85,B 0,C 180,E1 -9499.828,E2 -9499.828} C_VEL
LIN {X 0,Y 432.298,Z 360.249,A -85,B 0,C 180,E1 -9503.021,E2 -9503.021} C_VEL
LIN {X 0,Y 432.359,Z 360.251,A -85,B 0,C 180,E1 -9505.997,E2 -9505.997} C_VEL
LIN {X 0,Y 432.346,Z 360.235,A -85,B 0,C 180,E1 -9509.49,E2 -9509.49} C_VEL
LIN {X 0,Y 432.343,Z 360.253,A -85,B 0,C 180,E1 -9511.874,E2 -9511.874} C_VEL
LIN {X 0,Y 432.377,Z 360.249,A -85,B 0,C 180,E1 -9515.539,E2 -9515.539} C_VEL
LIN {X 0,Y 432.35,Z 360.252,A -85,B 0,C 180,E1 -9519.046,E2 -9519.046} C_VEL
LIN {X 0,Y 432.358,Z 360.252,A -85,B 0,C 180,E1 -9522.011,E2 -9522.011} C_VEL
LIN {X 0,Y 432.389,Z 360.248,A -85,B 0,C 180,E1 -9524.927,E2 -9524.927} C_VEL
LIN {X 0,Y 432.46,Z 360.235,A -85,B 0,C 180,E1 -9527.804,E2 -9527.804} C_VEL
LIN {X 0,Y 432.465,Z 360.233,A -85,B 0,C 180,E1 -9531.59,E2 -9531.59} C_VEL
LIN {X 0,Y 432.579,Z 360.227,A -85,B 0,C 180,E1 -9534.406,E2 -9534.406} C_VEL
LIN {X 0,Y 432.604,Z 360.224,A -85,B 0,C 180,E1 -9538.138,E2 -9538.138} C_VEL
LIN {X 0,Y 432.662,Z 360.209,A -85,B 0,C 180,E1 -9540,E2 -9540} C_VEL
LIN {X 0,Y 432.579,Z 360.221,A -85,B 0,C 180,E1 -9542.794,E2 -9542.794} C_VEL
LIN {X 0,Y 432.58,Z 360.223,A -85,B 0,C 180,E1 -9545.595,E2 -9545.595} C_VEL
LIN {X 0,Y 432.465,Z 360.239,A -85,B 0,C 180,E1 -9548.411,E2 -9548.411} C_VEL
LIN {X 0,Y 432.461,Z 360.238,A -85,B 0,C 180,E1 -9552.197,E2 -9552.197} C_VEL
LIN {X 0,Y 432.433,Z 360.242,A -85,B 0,C 180,E1 -9556.039,E2 -9556.039} C_VEL
LIN {X 0,Y 432.389,Z 360.229,A -85,B 0,C 180,E1 -9559.485,E2 -9559.485} C_VEL
LIN {X 0,Y 432.319,Z 360.257,A -85,B 0,C 180,E1 -9562.965,E2 -9562.965} C_VEL
LIN {X 0,Y 432.322,Z 360.241,A -85,B 0,C 180,E1 -9566.036,E2 -9566.036} C_VEL
LIN {X 0,Y 432.335,Z 360.253,A -85,B 0,C 180,E1 -9569.189,E2 -9569.189} C_VEL
LIN {X 0,Y 432.326,Z 360.254,A -85,B 0,C 180,E1 -9572.443,E2 -9572.443} C_VEL
LIN {X 0,Y 432.344,Z 360.242,A -85,B 0,C 180,E1 -9575.632,E2 -9575.632} C_VEL
LIN {X 0,Y 432.322,Z 360.252,A -85,B 0,C 180,E1 -9578.711,E2 -9578.711} C_VEL
LIN {X 0,Y 432.312,Z 360.258,A -85,B 0,C 180,E1 -9581.8,E2 -9581.8} C_VEL
LIN {X 0,Y 432.337,Z 360.259,A -85,B 0,C 180,E1 -9584.348,E2 -9584.348} C_VEL
LIN {X 0,Y 432.32,Z 360.257,A -85,B 0,C 180,E1 -9587.017,E2 -9587.017} C_VEL
LIN {X 0,Y 432.317,Z 360.261,A -85,B 0,C 180,E1 -9589.824,E2 -9589.824} C_VEL
LIN {X 0,Y 432.346,Z 360.305,A -85,B 0,C 180,E1 -9590.901,E2 -9590.901} C_VEL
LIN {X 0,Y 435.321,Z 372.183,A -85,B 0,C 180,E1 -9593.472,E2 -9593.472} C_VEL
LIN {X 0,Y 442.523,Z 388.279,A -85,B 0,C 180,E1 -9594.285,E2 -9594.285} C_VEL
LIN {X 0,Y 444.501,Z 397.792,A -85,B 0,C 180,E1 -9594.594,E2 -9594.594} C_VEL
LIN {X 0,Y 442.143,Z 526.778,A -85,B 0,C 180,E1 -9596.743,E2 -9596.743} C_VEL
LIN {X 0,Y 441.9,Z 542.755,A -85,B 0,C 180,E1 -9597.097,E2 -9597.097} C_VEL
LIN {X 0,Y 441.243,Z 556.909,A -85,B 0,C 180,E1 -9597.565,E2 -9597.565} C_VEL
LIN {X 0,Y 440.384,Z 571.301,A -85,B 0,C 180,E1 -9598.221,E2 -9598.221} C_VEL
LIN {X 0,Y 439.384,Z 585.699,A -85,B 0,C 180,E1 -9599.08,E2 -9599.08} C_VEL
LIN {X 0,Y 438.303,Z 599.275,A -85,B 0,C 180,E1 -9600.098,E2 -9600.098} C_VEL
LIN {X 0,Y 437.075,Z 612.276,A -85,B 0,C 180,E1 -9601.29,E2 -9601.29} C_VEL
LIN {X 0,Y 435.976,Z 623.811,A -85,B 0,C 180,E1 -9602.57,E2 -9602.57} C_VEL
LIN {X 0,Y 435.018,Z 633.79,A -85,B 0,C 180,E1 -9603.881,E2 -9603.881} C_VEL
LIN {X 0,Y 433.964,Z 643.735,A -85,B 0,C 180,E1 -9605.426,E2 -9605.426} C_VEL
LIN {X 0,Y 433.035,Z 647.351,A -85,B 0,C 180,E1 -9606.039,E2 -9606.039} C_VEL
LIN {X 0,Y 429.712,Z 652.991,A -85,B 0,C 180,E1 -9607.023,E2 -9607.023} C_VEL
LIN {X 0,Y 426.352,Z 658.24,A -85,B 0,C 180,E1 -9608.058,E2 -9608.058} C_VEL
LIN {X 0,Y 425.382,Z 661.075,A -85,B 0,C 180,E1 -9608.744,E2 -9608.744} C_VEL
LIN {X 0,Y 424.829,Z 667.785,A -85,B 0,C 180,E1 -9610.679,E2 -9610.679} C_VEL
LIN {X 0,Y 424.452,Z 673.147,A -85,B 0,C 180,E1 -9612.66,E2 -9612.66} C_VEL
LIN {X 0,Y 424.235,Z 677.099,A -85,B 0,C 180,E1 -9614.629,E2 -9614.629} C_VEL
LIN {X 0,Y 424.103,Z 679.732,A -85,B 0,C 180,E1 -9616.585,E2 -9616.585} C_VEL
LIN {X 0,Y 424.094,Z 681.146,A -85,B 0,C 180,E1 -9618.53,E2 -9618.53} C_VEL
LIN {X 0,Y 423.981,Z 681.398,A -85,B 0,C 180,E1 -9620.459,E2 -9620.459} C_VEL
LIN {X 0,Y 424.075,Z 680.501,A -85,B 0,C 180,E1 -9622.381,E2 -9622.381} C_VEL
LIN {X 0,Y 424.214,Z 678.459,A -85,B 0,C 180,E1 -9624.295,E2 -9624.295} C_VEL
LIN {X 0,Y 424.336,Z 675.221,A -85,B 0,C 180,E1 -9626.201,E2 -9626.201} C_VEL
LIN {X 0,Y 424.503,Z 670.715,A -85,B 0,C 180,E1 -9628.103,E2 -9628.103} C_VEL
LIN {X 0,Y 424.847,Z 664.876,A -85,B 0,C 180,E1 -9630,E2 -9630} C_VEL
LIN {X 0,Y 425.48,Z 657.537,A -85,B 0,C 180,E1 -9631.893,E2 -9631.893} C_VEL
LIN {X 0,Y 426.17,Z 649.698,A -85,B 0,C 180,E1 -9633.546,E2 -9633.546} C_VEL
LIN {X 0,Y 427.039,Z 640.318,A -85,B 0,C 180,E1 -9635.193,E2 -9635.193} C_VEL
LIN {X 0,Y 427.972,Z 630.78,A -85,B 0,C 180,E1 -9636.601,E2 -9636.601} C_VEL
LIN {X 0,Y 429.07,Z 619.476,A -85,B 0,C 180,E1 -9638.003,E2 -9638.003} C_VEL
LIN {X 0,Y 430.161,Z 607.072,A -85,B 0,C 180,E1 -9639.285,E2 -9639.285} C_VEL
LIN {X 0,Y 431.159,Z 594.911,A -85,B 0,C 180,E1 -9640.329,E2 -9640.329} C_VEL
LIN {X 0,Y 432.175,Z 581.75,A -85,B 0,C 180,E1 -9641.253,E2 -9641.253} C_VEL
LIN {X 0,Y 433.114,Z 567.234,A -85,B 0,C 180,E1 -9642.059,E2 -9642.059} C_VEL
LIN {X 0,Y 433.87,Z 552.114,A -85,B 0,C 180,E1 -9642.691,E2 -9642.691} C_VEL
LIN {X 0,Y 434.357,Z 536.246,A -85,B 0,C 180,E1 -9643.149,E2 -9643.149} C_VEL
LIN {X 0,Y 436.621,Z 397.981,A -85,B 0,C 180,E1 -9645.473,E2 -9645.473} C_VEL
LIN {X 0,Y 433.906,Z 387.075,A -85,B 0,C 180,E1 -9645.822,E2 -9645.822} C_VEL
LIN {X 0,Y 427.796,Z 371.807,A -85,B 0,C 180,E1 -9646.466,E2 -9646.466} C_VEL
LIN {X 0,Y 425.342,Z 361.13,A -85,B 0,C 180,E1 -9648.703,E2 -9648.703} C_VEL
LIN {X 0,Y 425.292,Z 361.134,A -85,B 0,C 180,E1 -9652.339,E2 -9652.339} C_VEL
LIN {X 0,Y 425.264,Z 361.138,A -85,B 0,C 180,E1 -9655.447,E2 -9655.447} C_VEL
LIN {X 0,Y 425.312,Z 361.13,A -85,B 0,C 180,E1 -9658.86,E2 -9658.86} C_VEL
LIN {X 0,Y 425.269,Z 361.131,A -85,B 0,C 180,E1 -9661.927,E2 -9661.927} C_VEL
LIN {X 0,Y 425.301,Z 361.133,A -85,B 0,C 180,E1 -9665.336,E2 -9665.336} C_VEL
LIN {X 0,Y 425.28,Z 361.133,A -85,B 0,C 180,E1 -9668.901,E2 -9668.901} C_VEL
LIN {X 0,Y 425.26,Z 361.134,A -85,B 0,C 180,E1 -9672.655,E2 -9672.655} C_VEL
LIN {X 0,Y 425.289,Z 361.128,A -85,B 0,C 180,E1 -9675.283,E2 -9675.283} C_VEL
LIN {X 0,Y 425.255,Z 361.135,A -85,B 0,C 180,E1 -9678.618,E2 -9678.618} C_VEL
LIN {X 0,Y 425.28,Z 361.131,A -85,B 0,C 180,E1 -9681.099,E2 -9681.099} C_VEL
LIN {X 0,Y 425.297,Z 361.129,A -85,B 0,C 180,E1 -9684.663,E2 -9684.663} C_VEL
LIN {X 0,Y 425.266,Z 361.137,A -85,B 0,C 180,E1 -9688.073,E2 -9688.073} C_VEL
LIN {X 0,Y 425.308,Z 361.12,A -85,B 0,C 180,E1 -9691.366,E2 -9691.366} C_VEL
LIN {X 0,Y 425.262,Z 361.109,A -85,B 0,C 180,E1 -9694.552,E2 -9694.552} C_VEL
LIN {X 0,Y 425.295,Z 361.132,A -85,B 0,C 180,E1 -9697.729,E2 -9697.729} C_VEL
LIN {X 0,Y 425.364,Z 361.12,A -85,B 0,C 180,E1 -9700.704,E2 -9700.704} C_VEL
LIN {X 0,Y 425.391,Z 361.118,A -85,B 0,C 180,E1 -9703.688,E2 -9703.688} C_VEL
LIN {X 0,Y 425.415,Z 361.111,A -85,B 0,C 180,E1 -9707.598,E2 -9707.598} C_VEL
LIN {X 0,Y 425.409,Z 361.119,A -85,B 0,C 180,E1 -9711.449,E2 -9711.449} C_VEL
LIN {X 0,Y 425.514,Z 361.094,A -85,B 0,C 180,E1 -9714.312,E2 -9714.312} C_VEL
LIN {X 0,Y 425.567,Z 361.097,A -85,B 0,C 180,E1 -9718.107,E2 -9718.107} C_VEL
LIN {X 0,Y 425.613,Z 361.087,A -85,B 0,C 180,E1 -9720,E2 -9720} C_VEL
LIN {X 0,Y 425.537,Z 361.095,A -85,B 0,C 180,E1 -9722.84,E2 -9722.84} C_VEL
LIN {X 0,Y 425.529,Z 361.105,A -85,B 0,C 180,E1 -9725.687,E2 -9725.687} C_VEL
LIN {X 0,Y 425.41,Z 361.111,A -85,B 0,C 180,E1 -9728.55,E2 -9728.55} C_VEL
LIN {X 0,Y 425.414,Z 361.109,A -85,B 0,C 180,E1 -9732.401,E2 -9732.401} C_VEL
LIN {X 0,Y 425.306,Z 361.13,A -85,B 0,C 180,E1 -9735.331,E2 -9735.331} C_VEL
LIN {X 0,Y 425.315,Z 361.123,A -85,B 0,C 180,E1 -9738.298,E2 -9738.298} C_VEL
LIN {X 0,Y 425.294,Z 361.132,A -85,B 0,C 180,E1 -9741.318,E2 -9741.318} C_VEL
LIN {X 0,Y 425.318,Z 361.126,A -85,B 0,C 180,E1 -9744.656,E2 -9744.656} C_VEL
LIN {X 0,Y 425.261,Z 361.138,A -85,B 0,C 180,E1 -9747.564,E2 -9747.564} C_VEL
LIN {X 0,Y 425.291,Z 361.13,A -85,B 0,C 180,E1 -9750.761,E2 -9750.761} C_VEL
LIN {X 0,Y 425.31,Z 361.129,A -85,B 0,C 180,E1 -9754.287,E2 -9754.287} C_VEL
LIN {X 0,Y 425.27,Z 361.136,A -85,B 0,C 180,E1 -9757.695,E2 -9757.695} C_VEL
LIN {X 0,Y 425.242,Z 361.135,A -85,B 0,C 180,E1 -9760.514,E2 -9760.514} C_VEL
LIN {X 0,Y 425.246,Z 361.139,A -85,B 0,C 180,E1 -9763.349,E2 -9763.349} C_VEL
LIN {X 0,Y 425.257,Z 361.14,A -85,B 0,C 180,E1 -9766.043,E2 -9766.043} C_VEL
LIN {X 0,Y 425.25,Z 361.139,A -85,B 0,C 180,E1 -9768.618,E2 -9768.618} C_VEL
LIN {X 0,Y 425.277,Z 361.138,A -85,B 0,C 180,E1 -9771.099,E2 -9771.099} C_VEL
LIN {X 0,Y 425.296,Z 361.133,A -85,B 0,C 180,E1 -9774.664,E2 -9774.664} C_VEL
LIN {X 0,Y 425.322,Z 361.302,A -85,B 0,C 180,E1 -9777.748,E2 -9777.748} C_VEL
LIN {X 0,Y 429.003,Z 376.405,A -85,B 0,C 180,E1 -9780.563,E2 -9780.563} C_VEL
LIN {X 0,Y 430.803,Z 384.475,A -85,B 0,C 180,E1 -9782.01,E2 -9782.01} C_VEL
LIN {X 0,Y 430.791,Z 389.412,A -85,B 0,C 180,E1 -9782.819,E2 -9782.819} C_VEL
LIN {X 0,Y 430.406,Z 395.006,A -85,B 0,C 180,E1 -9783.711,E2 -9783.711} C_VEL
LIN {X 0,Y 436.256,Z 426.471,A -85,B 0,C 180,E1 -9784.609,E2 -9784.609} C_VEL
LIN {X 0,Y 434.177,Z 561.616,A -85,B 0,C 180,E1 -9786.888,E2 -9786.888} C_VEL
LIN {X 0,Y 433.498,Z 577.336,A -85,B 0,C 180,E1 -9787.337,E2 -9787.337} C_VEL
LIN {X 0,Y 432.644,Z 592.623,A -85,B 0,C 180,E1 -9787.975,E2 -9787.975} C_VEL
LIN {X 0,Y 431.67,Z 606.846,A -85,B 0,C 180,E1 -9788.761,E2 -9788.761} C_VEL
LIN {X 0,Y 430.603,Z 620.369,A -85,B 0,C 180,E1 -9789.706,E2 -9789.706} C_VEL
LIN {X 0,Y 429.374,Z 634.109,A -85,B 0,C 180,E1 -9790.891,E2 -9790.891} C_VEL
LIN {X 0,Y 428.34,Z 645.709,A -85,B 0,C 180,E1 -9792.107,E2 -9792.107} C_VEL
LIN {X 0,Y 427.322,Z 657.006,A -85,B 0,C 180,E1 -9793.518,E2 -9793.518} C_VEL
LIN {X 0,Y 426.407,Z 666.679,A -85,B 0,C 180,E1 -9794.954,E2 -9794.954} C_VEL
LIN {X 0,Y 425.584,Z 676.178,A -85,B 0,C 180,E1 -9796.633,E2 -9796.633} C_VEL
LIN {X 0,Y 425.057,Z 684.08,A -85,B 0,C 180,E1 -9798.314,E2 -9798.314} C_VEL
LIN {X 0,Y 424.587,Z 690.625,A -85,B 0,C 180,E1 -9799.991,E2 -9799.991} C_VEL
LIN {X 0,Y 424.346,Z 696.636,A -85,B 0,C 180,E1 -9801.907,E2 -9801.907} C_VEL
LIN {X 0,Y 424.174,Z 701.18,A -85,B 0,C 180,E1 -9803.782,E2 -9803.782} C_VEL
LIN {X 0,Y 424.143,Z 703.816,A -85,B 0,C 180,E1 -9805.248,E2 -9805.248} C_VEL
LIN {X 0,Y 424.124,Z 706.217,A -85,B 0,C 180,E1 -9807.15,E2 -9807.15} C_VEL
LIN {X 0,Y 424.087,Z 707.447,A -85,B 0,C 180,E1 -9809.05,E2 -9809.05} C_VEL
LIN {X 0,Y 424.087,Z 707.475,A -85,B 0,C 180,E1 -9810.95,E2 -9810.95} C_VEL
LIN {X 0,Y 424.123,Z 706.359,A -85,B 0,C 180,E1 -9812.849,E2 -9812.849} C_VEL
LIN {X 0,Y 424.12,Z 704.092,A -85,B 0,C 180,E1 -9814.753,E2 -9814.753} C_VEL
LIN {X 0,Y 424.209,Z 700.633,A -85,B 0,C 180,E1 -9816.66,E2 -9816.66} C_VEL
LIN {X 0,Y 424.396,Z 695.897,A -85,B 0,C 180,E1 -9818.571,E2 -9818.571} C_VEL
LIN {X 0,Y 424.714,Z 689.753,A -85,B 0,C 180,E1 -9820.488,E2 -9820.488} C_VEL
LIN {X 0,Y 425.229,Z 683.081,A -85,B 0,C 180,E1 -9822.165,E2 -9822.165} C_VEL
LIN {X 0,Y 426.029,Z 673.845,A -85,B 0,C 180,E1 -9824.083,E2 -9824.083} C_VEL
LIN {X 0,Y 426.982,Z 664.014,A -85,B 0,C 180,E1 -9825.759,E2 -9825.759} C_VEL
LIN {X 0,Y 428.218,Z 652.591,A -85,B 0,C 180,E1 -9827.374,E2 -9827.374} C_VEL
LIN {X 0,Y 429.34,Z 641.016,A -85,B 0,C 180,E1 -9828.738,E2 -9828.738} C_VEL
LIN {X 0,Y 430.572,Z 628.945,A -85,B 0,C 180,E1 -9829.921,E2 -9829.921} C_VEL
LIN {X 0,Y 431.833,Z 615.87,A -85,B 0,C 180,E1 -9830.98,E2 -9830.98} C_VEL
LIN {X 0,Y 433.025,Z 601.537,A -85,B 0,C 180,E1 -9831.919,E2 -9831.919} C_VEL
LIN {X 0,Y 434.022,Z 587.533,A -85,B 0,C 180,E1 -9832.634,E2 -9832.634} C_VEL
LIN {X 0,Y 434.907,Z 572.663,A -85,B 0,C 180,E1 -9833.197,E2 -9833.197} C_VEL
LIN {X 0,Y 435.543,Z 556.579,A -85,B 0,C 180,E1 -9833.602,E2 -9833.602} C_VEL
LIN {X 0,Y 437.839,Z 427.075,A -85,B 0,C 180,E1 -9835.808,E2 -9835.808} C_VEL
LIN {X 0,Y 433.871,Z 406.213,A -85,B 0,C 180,E1 -9836.473,E2 -9836.473} C_VEL
LIN {X 0,Y 431.301,Z 394.577,A -85,B 0,C 180,E1 -9836.905,E2 -9836.905} C_VEL
LIN {X 0,Y 431.866,Z 388.542,A -85,B 0,C 180,E1 -9837.896,E2 -9837.896} C_VEL
LIN {X 0,Y 430.79,Z 382.38,A -85,B 0,C 180,E1 -9839.04,E2 -9839.04} C_VEL
LIN {X 0,Y 427.915,Z 370.679,A -85,B 0,C 180,E1 -9841.347,E2 -9841.347} C_VEL
LIN {X 0,Y 425.303,Z 361.135,A -85,B 0,C 180,E1 -9843.329,E2 -9843.329} C_VEL
LIN {X 0,Y 425.26,Z 361.133,A -85,B 0,C 180,E1 -9846.509,E2 -9846.509} C_VEL
LIN {X 0,Y 425.257,Z 361.131,A -85,B 0,C 180,E1 -9849.037,E2 -9849.037} C_VEL
LIN {X 0,Y 425.259,Z 361.134,A -85,B 0,C 180,E1 -9852.655,E2 -9852.655} C_VEL
LIN {X 0,Y 425.283,Z 361.134,A -85,B 0,C 180,E1 -9855.283,E2 -9855.283} C_VEL
LIN {X 0,Y 425.247,Z 361.141,A -85,B 0,C 180,E1 -9858.618,E2 -9858.618} C_VEL
LIN {X 0,Y 425.275,Z 361.134,A -85,B 0,C 180,E1 -9861.099,E2 -9861.099} C_VEL
LIN {X 0,Y 425.297,Z 361.123,A -85,B 0,C 180,E1 -9864.664,E2 -9864.664} C_VEL
LIN {X 0,Y 425.265,Z 361.127,A -85,B 0,C 180,E1 -9868.073,E2 -9868.073} C_VEL
LIN {X 0,Y 425.31,Z 361.127,A -85,B 0,C 180,E1 -9871.367,E2 -9871.367} C_VEL
LIN {X 0,Y 425.271,Z 361.137,A -85,B 0,C 180,E1 -9874.553,E2 -9874.553} C_VEL
LIN {X 0,Y 425.284,Z 361.131,A -85,B 0,C 180,E1 -9876.634,E2 -9876.634} C_VEL
LIN {X 0,Y 425.296,Z 361.131,A -85,B 0,C 180,E1 -9879.695,E2 -9879.695} C_VEL
LIN {X 0,Y 425.331,Z 361.128,A -85,B 0,C 180,E1 -9882.697,E2 -9882.697} C_VEL
LIN {X 0,Y 425.344,Z 361.124,A -85,B 0,C 180,E1 -9885.65,E2 -9885.65} C_VEL
LIN {X 0,Y 425.351,Z 361.125,A -85,B 0,C 180,E1 -9888.564,E2 -9888.564} C_VEL
LIN {X 0,Y 425.409,Z 361.111,A -85,B 0,C 180,E1 -9891.45,E2 -9891.45} C_VEL
LIN {X 0,Y 425.533,Z 361.106,A -85,B 0,C 180,E1 -9894.313,E2 -9894.313} C_VEL
LIN {X 0,Y 425.573,Z 361.099,A -85,B 0,C 180,E1 -9898.108,E2 -9898.108} C_VEL
LIN {X 0,Y 425.511,Z 361.106,A -85,B 0,C 180,E1 -9900.947,E2 -9900.947} C_VEL
LIN {X 0,Y 425.533,Z 361.098,A -85,B 0,C 180,E1 -9902.84,E2 -9902.84} C_VEL
LIN {X 0,Y 425.534,Z 361.101,A -85,B 0,C 180,E1 -9905.687,E2 -9905.687} C_VEL
LIN {X 0,Y 425.409,Z 361.12,A -85,B 0,C 180,E1 -9908.551,E2 -9908.551} C_VEL
LIN {X 0,Y 425.415,Z 361.119,A -85,B 0,C 180,E1 -9912.402,E2 -9912.402} C_VEL
LIN {X 0,Y 425.39,Z 361.123,A -85,B 0,C 180,E1 -9916.312,E2 -9916.312} C_VEL
LIN {X 0,Y 425.331,Z 361.107,A -85,B 0,C 180,E1 -9919.636,E2 -9919.636} C_VEL
LIN {X 0,Y 425.29,Z 361.133,A -85,B 0,C 180,E1 -9922.339,E2 -9922.339} C_VEL
LIN {X 0,Y 425.309,Z 361.119,A -85,B 0,C 180,E1 -9924.653,E2 -9924.653} C_VEL
LIN {X 0,Y 425.299,Z 361.128,A -85,B 0,C 180,E1 -9927.562,E2 -9927.562} C_VEL
LIN {X 0,Y 425.291,Z 361.121,A -85,B 0,C 180,E1 -9930.816,E2 -9930.816} C_VEL
LIN {X 0,Y 425.312,Z 361.129,A -85,B 0,C 180,E1 -9934.288,E2 -9934.288} C_VEL
LIN {X 0,Y 425.274,Z 361.135,A -85,B 0,C 180,E1 -9937.695,E2 -9937.695} C_VEL
LIN {X 0,Y 425.247,Z 361.139,A -85,B 0,C 180,E1 -9940.515,E2 -9940.515} C_VEL
LIN {X 0,Y 425.253,Z 361.139,A -85,B 0,C 180,E1 -9943.35,E2 -9943.35} C_VEL
LIN {X 0,Y 425.264,Z 361.135,A -85,B 0,C 180,E1 -9946.044,E2 -9946.044} C_VEL
LIN {X 0,Y 425.269,Z 361.139,A -85,B 0,C 180,E1 -9948.621,E2 -9948.621} C_VEL
LIN {X 0,Y 425.292,Z 361.238,A -85,B 0,C 180,E1 -9950.451,E2 -9950.451} C_VEL
LIN {X 0,Y 428.088,Z 372.211,A -85,B 0,C 180,E1 -9952.923,E2 -9952.923} C_VEL
LIN {X 0,Y 436.461,Z 390.686,A -85,B 0,C 180,E1 -9953.899,E2 -9953.899} C_VEL
LIN {X 0,Y 438.217,Z 398.187,A -85,B 0,C 180,E1 -9954.162,E2 -9954.162} C_VEL
LIN {X 0,Y 435.823,Z 524.547,A -85,B 0,C 180,E1 -9956.301,E2 -9956.301} C_VEL
LIN {X 0,Y 435.547,Z 541.394,A -85,B 0,C 180,E1 -9956.658,E2 -9956.658} C_VEL
LIN {X 0,Y 434.809,Z 556.404,A -85,B 0,C 180,E1 -9957.144,E2 -9957.144} C_VEL
LIN {X 0,Y 433.945,Z 571.324,A -85,B 0,C 180,E1 -9957.83,E2 -9957.83} C_VEL
LIN {X 0,Y 433.032,Z 583.913,A -85,B 0,C 180,E1 -9958.575,E2 -9958.575} C_VEL
LIN {X 0,Y 431.878,Z 597.761,A -85,B 0,C 180,E1 -9959.597,E2 -9959.597} C_VEL
LIN {X 0,Y 430.685,Z 609.931,A -85,B 0,C 180,E1 -9960.689,E2 -9960.689} C_VEL
LIN {X 0,Y 429.461,Z 621.843,A -85,B 0,C 180,E1 -9961.979,E2 -9961.979} C_VEL
LIN {X 0,Y 428.293,Z 633.062,A -85,B 0,C 180,E1 -9963.439,E2 -9963.439} C_VEL
LIN {X 0,Y 427.229,Z 642.493,A -85,B 0,C 180,E1 -9964.899,E2 -9964.899} C_VEL
LIN {X 0,Y 426.247,Z 652.132,A -85,B 0,C 180,E1 -9966.689,E2 -9966.689} C_VEL
LIN {X 0,Y 425.515,Z 659.863,A -85,B 0,C 180,E1 -9968.439,E2 -9968.439} C_VEL
LIN {X 0,Y 425.382,Z 661.075,A -85,B 0,C 180,E1 -9968.744,E2 -9968.744} C_VEL
LIN {X 0,Y 424.46,Z 663.79,A -85,B 0,C 180,E1 -9969.446,E2 -9969.446} C_VEL
LIN {X 0,Y 421.292,Z 667.916,A -85,B 0,C 180,E1 -9970.589,E2 -9970.589} C_VEL
LIN {X 0,Y 418.195,Z 671.57,A -85,B 0,C 180,E1 -9971.775,E2 -9971.775} C_VEL
LIN {X 0,Y 417.395,Z 673.436,A -85,B 0,C 180,E1 -9972.537,E2 -9972.537} C_VEL
LIN {X 0,Y 417.183,Z 677.07,A -85,B 0,C 180,E1 -9974.363,E2 -9974.363} C_VEL
LIN {X 0,Y 417.017,Z 679.792,A -85,B 0,C 180,E1 -9976.353,E2 -9976.353} C_VEL
LIN {X 0,Y 417.01,Z 681.298,A -85,B 0,C 180,E1 -9978.332,E2 -9978.332} C_VEL
LIN {X 0,Y 416.887,Z 681.64,A -85,B 0,C 180,E1 -9980.295,E2 -9980.295} C_VEL
LIN {X 0,Y 416.973,Z 680.834,A -85,B 0,C 180,E1 -9982.251,E2 -9982.251} C_VEL
LIN {X 0,Y 417.125,Z 678.873,A -85,B 0,C 180,E1 -9984.198,E2 -9984.198} C_VEL
LIN {X 0,Y 417.23,Z 675.692,A -85,B 0,C 180,E1 -9986.137,E2 -9986.137} C_VEL
LIN {X 0,Y 417.441,Z 671.278,A -85,B 0,C 180,E1 -9988.07,E2 -9988.07} C_VEL
LIN {X 0,Y 417.763,Z 665.542,A -85,B 0,C 180,E1 -9990,E2 -9990} C_VEL
LIN {X 0,Y 418.413,Z 658.312,A -85,B 0,C 180,E1 -9991.925,E2 -9991.925} C_VEL
LIN {X 0,Y 419.137,Z 650.59,A -85,B 0,C 180,E1 -9993.605,E2 -9993.605} C_VEL
LIN {X 0,Y 420.028,Z 641.345,A -85,B 0,C 180,E1 -9995.28,E2 -9995.28} C_VEL
LIN {X 0,Y 421.003,Z 631.961,A -85,B 0,C 180,E1 -9996.711,E2 -9996.711} C_VEL
LIN {X 0,Y 422.128,Z 620.844,A -85,B 0,C 180,E1 -9998.136,E2 -9998.136} C_VEL
LIN {X 0,Y 423.259,Z 608.672,A -85,B 0,C 180,E1 -9999.437,E2 -9999.437} C_VEL
LIN {X 0,Y 424.415,Z 595.261,A -85,B 0,C 180,E1 -10000.616,E2 -10000.616} C_VEL
LIN {X 0,Y 425.467,Z 582.115,A -85,B 0,C 180,E1 -10001.554,E2 -10001.554} C_VEL
LIN {X 0,Y 426.427,Z 567.639,A -85,B 0,C 180,E1 -10002.372,E2 -10002.372} C_VEL
LIN {X 0,Y 427.21,Z 552.582,A -85,B 0,C 180,E1 -10003.013,E2 -10003.013} C_VEL
LIN {X 0,Y 427.72,Z 536.739,A -85,B 0,C 180,E1 -10003.481,E2 -10003.481} C_VEL
LIN {X 0,Y 430.076,Z 399.442,A -85,B 0,C 180,E1 -10005.823,E2 -10005.823} C_VEL
LIN {X 0,Y 427.762,Z 389.734,A -85,B 0,C 180,E1 -10006.134,E2 -10006.134} C_VEL
LIN {X 0,Y 420.597,Z 372.036,A -85,B 0,C 180,E1 -10006.9,E2 -10006.9} C_VEL
LIN {X 0,Y 418.316,Z 362.005,A -85,B 0,C 180,E1 -10009.06,E2 -10009.06} C_VEL
LIN {X 0,Y 418.233,Z 362.014,A -85,B 0,C 180,E1 -10012.737,E2 -10012.737} C_VEL
LIN {X 0,Y 418.23,Z 362.014,A -85,B 0,C 180,E1 -10015.907,E2 -10015.907} C_VEL
LIN {X 0,Y 418.263,Z 362.008,A -85,B 0,C 180,E1 -10019.162,E2 -10019.162} C_VEL
LIN {X 0,Y 418.262,Z 362.002,A -85,B 0,C 180,E1 -10022.844,E2 -10022.844} C_VEL
LIN {X 0,Y 418.244,Z 362.004,A -85,B 0,C 180,E1 -10026.237,E2 -10026.237} C_VEL
LIN {X 0,Y 418.202,Z 362.011,A -85,B 0,C 180,E1 -10029.688,E2 -10029.688} C_VEL
LIN {X 0,Y 418.211,Z 362.013,A -85,B 0,C 180,E1 -10032.317,E2 -10032.317} C_VEL
LIN {X 0,Y 418.24,Z 362.008,A -85,B 0,C 180,E1 -10035.108,E2 -10035.108} C_VEL
LIN {X 0,Y 418.227,Z 362.013,A -85,B 0,C 180,E1 -10037.764,E2 -10037.764} C_VEL
LIN {X 0,Y 418.238,Z 362.01,A -85,B 0,C 180,E1 -10041.556,E2 -10041.556} C_VEL
LIN {X 0,Y 418.254,Z 362.009,A -85,B 0,C 180,E1 -10045.158,E2 -10045.158} C_VEL
LIN {X 0,Y 418.246,Z 362.012,A -85,B 0,C 180,E1 -10047.471,E2 -10047.471} C_VEL
LIN {X 0,Y 418.265,Z 362.002,A -85,B 0,C 180,E1 -10050.897,E2 -10050.897} C_VEL
LIN {X 0,Y 418.221,Z 361.983,A -85,B 0,C 180,E1 -10054.092,E2 -10054.092} C_VEL
LIN {X 0,Y 418.231,Z 362.005,A -85,B 0,C 180,E1 -10057.263,E2 -10057.263} C_VEL
LIN {X 0,Y 418.286,Z 362.002,A -85,B 0,C 180,E1 -10060.364,E2 -10060.364} C_VEL
LIN {X 0,Y 418.32,Z 361.994,A -85,B 0,C 180,E1 -10063.404,E2 -10063.404} C_VEL
LIN {X 0,Y 418.35,Z 361.994,A -85,B 0,C 180,E1 -10066.999,E2 -10066.999} C_VEL
LIN {X 0,Y 418.338,Z 361.994,A -85,B 0,C 180,E1 -10070.328,E2 -10070.328} C_VEL
LIN {X 0,Y 418.444,Z 361.985,A -85,B 0,C 180,E1 -10073.248,E2 -10073.248} C_VEL
LIN {X 0,Y 418.319,Z 361.991,A -85,B 0,C 180,E1 -10075.181,E2 -10075.181} C_VEL
LIN {X 0,Y 418.536,Z 361.973,A -85,B 0,C 180,E1 -10078.075,E2 -10078.075} C_VEL
LIN {X 0,Y 418.565,Z 361.965,A -85,B 0,C 180,E1 -10080,E2 -10080} C_VEL
LIN {X 0,Y 418.492,Z 361.972,A -85,B 0,C 180,E1 -10082.887,E2 -10082.887} C_VEL
LIN {X 0,Y 418.487,Z 361.98,A -85,B 0,C 180,E1 -10085.783,E2 -10085.783} C_VEL
LIN {X 0,Y 418.379,Z 361.987,A -85,B 0,C 180,E1 -10088.695,E2 -10088.695} C_VEL
LIN {X 0,Y 418.316,Z 362,A -85,B 0,C 180,E1 -10091.631,E2 -10091.631} C_VEL
LIN {X 0,Y 418.28,Z 362.001,A -85,B 0,C 180,E1 -10094.597,E2 -10094.597} C_VEL
LIN {X 0,Y 418.258,Z 362.004,A -85,B 0,C 180,E1 -10097.605,E2 -10097.605} C_VEL
LIN {X 0,Y 418.251,Z 362.005,A -85,B 0,C 180,E1 -10100.663,E2 -10100.663} C_VEL
LIN {X 0,Y 418.274,Z 362.009,A -85,B 0,C 180,E1 -10103.782,E2 -10103.782} C_VEL
LIN {X 0,Y 418.216,Z 362.01,A -85,B 0,C 180,E1 -10107.044,E2 -10107.044} C_VEL
LIN {X 0,Y 418.242,Z 362.009,A -85,B 0,C 180,E1 -10110.272,E2 -10110.272} C_VEL
LIN {X 0,Y 418.248,Z 362.012,A -85,B 0,C 180,E1 -10113.677,E2 -10113.677} C_VEL
LIN {X 0,Y 418.233,Z 362.012,A -85,B 0,C 180,E1 -10117.225,E2 -10117.225} C_VEL
LIN {X 0,Y 418.206,Z 362.012,A -85,B 0,C 180,E1 -10120.867,E2 -10120.867} C_VEL
LIN {X 0,Y 418.202,Z 362.019,A -85,B 0,C 180,E1 -10123.728,E2 -10123.728} C_VEL
LIN {X 0,Y 418.201,Z 362.016,A -85,B 0,C 180,E1 -10126.447,E2 -10126.447} C_VEL
LIN {X 0,Y 418.207,Z 362.018,A -85,B 0,C 180,E1 -10129.132,E2 -10129.132} C_VEL
LIN {X 0,Y 418.234,Z 362.013,A -85,B 0,C 180,E1 -10132.775,E2 -10132.775} C_VEL
LIN {X 0,Y 418.247,Z 362.012,A -85,B 0,C 180,E1 -10136.322,E2 -10136.322} C_VEL
LIN {X 0,Y 418.269,Z 362.16,A -85,B 0,C 180,E1 -10137.389,E2 -10137.389} C_VEL
LIN {X 0,Y 421.971,Z 377.321,A -85,B 0,C 180,E1 -10140.271,E2 -10140.271} C_VEL
LIN {X 0,Y 424.108,Z 387.663,A -85,B 0,C 180,E1 -10142.148,E2 -10142.148} C_VEL
LIN {X 0,Y 423.654,Z 394.805,A -85,B 0,C 180,E1 -10143.31,E2 -10143.31} C_VEL
LIN {X 0,Y 429.77,Z 427.985,A -85,B 0,C 180,E1 -10144.271,E2 -10144.271} C_VEL
LIN {X 0,Y 427.567,Z 561.032,A -85,B 0,C 180,E1 -10146.541,E2 -10146.541} C_VEL
LIN {X 0,Y 426.849,Z 576.72,A -85,B 0,C 180,E1 -10146.989,E2 -10146.989} C_VEL
LIN {X 0,Y 426.028,Z 591.685,A -85,B 0,C 180,E1 -10147.616,E2 -10147.616} C_VEL
LIN {X 0,Y 425.009,Z 606.031,A -85,B 0,C 180,E1 -10148.412,E2 -10148.412} C_VEL
LIN {X 0,Y 423.879,Z 619.66,A -85,B 0,C 180,E1 -10149.37,E2 -10149.37} C_VEL
LIN {X 0,Y 422.575,Z 633.506,A -85,B 0,C 180,E1 -10150.572,E2 -10150.572} C_VEL
LIN {X 0,Y 421.388,Z 646.226,A -85,B 0,C 180,E1 -10151.926,E2 -10151.926} C_VEL
LIN {X 0,Y 420.257,Z 658.289,A -85,B 0,C 180,E1 -10153.483,E2 -10153.483} C_VEL
LIN {X 0,Y 419.334,Z 667.75,A -85,B 0,C 180,E1 -10154.943,E2 -10154.943} C_VEL
LIN {X 0,Y 418.479,Z 677.262,A -85,B 0,C 180,E1 -10156.694,E2 -10156.694} C_VEL
LIN {X 0,Y 417.964,Z 684.743,A -85,B 0,C 180,E1 -10158.359,E2 -10158.359} C_VEL
LIN {X 0,Y 417.445,Z 691.931,A -85,B 0,C 180,E1 -10160.308,E2 -10160.308} C_VEL
LIN {X 0,Y 417.231,Z 697.594,A -85,B 0,C 180,E1 -10162.255,E2 -10162.255} C_VEL
LIN {X 0,Y 417.057,Z 701.883,A -85,B 0,C 180,E1 -10164.197,E2 -10164.197} C_VEL
LIN {X 0,Y 416.99,Z 704.909,A -85,B 0,C 180,E1 -10166.134,E2 -10166.134} C_VEL
LIN {X 0,Y 417.065,Z 706.745,A -85,B 0,C 180,E1 -10168.069,E2 -10168.069} C_VEL
LIN {X 0,Y 417.001,Z 707.384,A -85,B 0,C 180,E1 -10170,E2 -10170} C_VEL
LIN {X 0,Y 417.065,Z 706.856,A -85,B 0,C 180,E1 -10171.931,E2 -10171.931} C_VEL
LIN {X 0,Y 416.988,Z 705.185,A -85,B 0,C 180,E1 -10173.866,E2 -10173.866} C_VEL
LIN {X 0,Y 417.057,Z 702.352,A -85,B 0,C 180,E1 -10175.803,E2 -10175.803} C_VEL
LIN {X 0,Y 417.216,Z 698.291,A -85,B 0,C 180,E1 -10177.745,E2 -10177.745} C_VEL
LIN {X 0,Y 417.482,Z 692.892,A -85,B 0,C 180,E1 -10179.691,E2 -10179.691} C_VEL
LIN {X 0,Y 418.075,Z 686.02,A -85,B 0,C 180,E1 -10181.638,E2 -10181.638} C_VEL
LIN {X 0,Y 418.721,Z 677.498,A -85,B 0,C 180,E1 -10183.591,E2 -10183.591} C_VEL
LIN {X 0,Y 419.63,Z 668.448,A -85,B 0,C 180,E1 -10185.295,E2 -10185.295} C_VEL
LIN {X 0,Y 420.8,Z 657.577,A -85,B 0,C 180,E1 -10186.994,E2 -10186.994} C_VEL
LIN {X 0,Y 422.175,Z 645.387,A -85,B 0,C 180,E1 -10188.565,E2 -10188.565} C_VEL
LIN {X 0,Y 423.509,Z 632.989,A -85,B 0,C 180,E1 -10189.889,E2 -10189.889} C_VEL
LIN {X 0,Y 424.891,Z 619.302,A -85,B 0,C 180,E1 -10191.085,E2 -10191.085} C_VEL
LIN {X 0,Y 426.154,Z 605.897,A -85,B 0,C 180,E1 -10192.036,E2 -10192.036} C_VEL
LIN {X 0,Y 427.324,Z 590.918,A -85,B 0,C 180,E1 -10192.872,E2 -10192.872} C_VEL
LIN {X 0,Y 428.319,Z 575.461,A -85,B 0,C 180,E1 -10193.511,E2 -10193.511} C_VEL
LIN {X 0,Y 429.108,Z 559.812,A -85,B 0,C 180,E1 -10193.946,E2 -10193.946} C_VEL
LIN {X 0,Y 431.533,Z 427.929,A -85,B 0,C 180,E1 -10196.238,E2 -10196.238} C_VEL
LIN {X 0,Y 427.151,Z 405.083,A -85,B 0,C 180,E1 -10196.992,E2 -10196.992} C_VEL
LIN {X 0,Y 424.728,Z 394.457,A -85,B 0,C 180,E1 -10197.387,E2 -10197.387} C_VEL
LIN {X 0,Y 425.116,Z 390.154,A -85,B 0,C 180,E1 -10198.11,E2 -10198.11} C_VEL
LIN {X 0,Y 423.311,Z 380.982,A -85,B 0,C 180,E1 -10199.873,E2 -10199.873} C_VEL
LIN {X 0,Y 420.125,Z 368.834,A -85,B 0,C 180,E1 -10202.365,E2 -10202.365} C_VEL
LIN {X 0,Y 418.255,Z 362.012,A -85,B 0,C 180,E1 -10203.858,E2 -10203.858} C_VEL
LIN {X 0,Y 418.234,Z 362.013,A -85,B 0,C 180,E1 -10207.225,E2 -10207.225} C_VEL
LIN {X 0,Y 418.206,Z 362.013,A -85,B 0,C 180,E1 -10210.867,E2 -10210.867} C_VEL
LIN {X 0,Y 418.203,Z 362.016,A -85,B 0,C 180,E1 -10213.729,E2 -10213.729} C_VEL
LIN {X 0,Y 418.199,Z 362.018,A -85,B 0,C 180,E1 -10216.448,E2 -10216.448} C_VEL
LIN {X 0,Y 418.206,Z 362.015,A -85,B 0,C 180,E1 -10219.133,E2 -10219.133} C_VEL
LIN {X 0,Y 418.233,Z 362.002,A -85,B 0,C 180,E1 -10222.776,E2 -10222.776} C_VEL
LIN {X 0,Y 418.248,Z 362.012,A -85,B 0,C 180,E1 -10226.323,E2 -10226.323} C_VEL
LIN {X 0,Y 418.242,Z 361.992,A -85,B 0,C 180,E1 -10229.728,E2 -10229.728} C_VEL
LIN {X 0,Y 418.244,Z 362.007,A -85,B 0,C 180,E1 -10233.019,E2 -10233.019} C_VEL
LIN {X 0,Y 418.273,Z 362.009,A -85,B 0,C 180,E1 -10236.218,E2 -10236.218} C_VEL
